LIN {X 768.326, Y -27.278, Z 404, A 0, B 90, C -0, E1 0, E2 0, E3 0, E4 0} C_DIS
LIN {X 766.132, Y -26.943, Z 404, A 0, B 90, C -0, E1 0, E2 0, E3 0, E4 0} C_DIS
LIN {X 763.95, Y -26.54, Z 404, A 0, B 90, C -0, E1 0, E2 0, E3 0, E4 0} C_DIS
LIN {X 761.781, Y -26.068, Z 404, A 0, B 90, C -0, E1 0, E2 0, E3 0, E4 0} C_DIS
LIN {X 759.629, Y -25.528, Z 404, A 0, B 90, C -0, E1 0, E2 0, E3 0, E4 0} C_DIS
LIN {X 757.494, Y -24.921, Z 404, A 0, B 90, C -0, E1 0, E2 0, E3 0, E4 0} C_DIS
LIN {X 755.379, Y -24.248, Z 404, A 0, B 90, C -0, E1 0, E2 0, E3 0, E4 0} C_DIS
LIN {X 753.287, Y -23.508, Z 404, A 0, B 90, C -0, E1 0, E2 0, E3 0, E4 0} C_DIS
LIN {X 751.219, Y -22.703, Z 404, A 0, B 90, C -0, E1 0, E2 0, E3 0, E4 0} C_DIS
LIN {X 749.177, Y -21.833, Z 404, A 0, B 90, C -0, E1 0, E2 0, E3 0, E4 0} C_DIS
LIN {X 747.163, Y -20.9, Z 404, A 0, B 90, C -0, E1 0, E2 0, E3 0, E4 0} C_DIS
LIN {X 745.18, Y -19.903, Z 404, A 0, B 90, C -0, E1 0, E2 0, E3 0, E4 0} C_DIS
LIN {X 743.229, Y -18.845, Z 404, A 0, B 90, C -0, E1 0, E2 0, E3 0, E4 0} C_DIS
LIN {X 741.313, Y -17.727, Z 404, A 0, B 90, C -0, E1 0, E2 0, E3 0, E4 0} C_DIS
LIN {X 739.432, Y -16.548, Z 404, A 0, B 90, C -0, E1 0, E2 0, E3 0, E4 0} C_DIS
LIN {X 737.589, Y -15.311, Z 404, A 0, B 90, C -0, E1 0, E2 0, E3 0, E4 0} C_DIS
LIN {X 735.786, Y -14.017, Z 404, A 0, B 90, C -0, E1 0, E2 0, E3 0, E4 0} C_DIS
LIN {X 734.025, Y -12.667, Z 404, A 0, B 90, C -0, E1 0, E2 0, E3 0, E4 0} C_DIS
LIN {X 732.307, Y -11.262, Z 404, A 0, B 90, C -0, E1 0, E2 0, E3 0, E4 0} C_DIS
LIN {X 730.634, Y -9.804, Z 404, A 0, B 90, C -0, E1 0, E2 0, E3 0, E4 0} C_DIS
LIN {X 729.007, Y -8.294, Z 404, A 0, B 90, C -0, E1 0, E2 0, E3 0, E4 0} C_DIS
LIN {X 727.429, Y -6.734, Z 404, A 0, B 90, C -0, E1 0, E2 0, E3 0, E4 0} C_DIS
LIN {X 725.901, Y -5.125, Z 404, A 0, B 90, C -0, E1 0, E2 0, E3 0, E4 0} C_DIS
LIN {X 724.423, Y -3.468, Z 404, A 0, B 90, C -0, E1 0, E2 0, E3 0, E4 0} C_DIS
LIN {X 722.999, Y -1.766, Z 404, A 0, B 90, C -0, E1 0, E2 0, E3 0, E4 0} C_DIS
LIN {X 721.629, Y -0.02, Z 404, A 0, B 90, C -0, E1 0, E2 0, E3 0, E4 0} C_DIS
LIN {X 720.314, Y 1.768, Z 404, A 0, B 90, C -0, E1 0, E2 0, E3 0, E4 0} C_DIS
LIN {X 719.056, Y 3.596, Z 404, A 0, B 90, C -0, E1 0, E2 0, E3 0, E4 0} C_DIS
LIN {X 717.856, Y 5.463, Z 404, A 0, B 90, C -0, E1 0, E2 0, E3 0, E4 0} C_DIS
LIN {X 716.715, Y 7.367, Z 404, A 0, B 90, C -0, E1 0, E2 0, E3 0, E4 0} C_DIS
LIN {X 715.635, Y 9.305, Z 404, A 0, B 90, C -0, E1 0, E2 0, E3 0, E4 0} C_DIS
LIN {X 714.616, Y 11.277, Z 404, A 0, B 90, C -0, E1 0, E2 0, E3 0, E4 0} C_DIS
LIN {X 713.66, Y 13.28, Z 404, A 0, B 90, C -0, E1 0, E2 0, E3 0, E4 0} C_DIS
LIN {X 712.767, Y 15.311, Z 404, A 0, B 90, C -0, E1 0, E2 0, E3 0, E4 0} C_DIS
LIN {X 711.938, Y 17.37, Z 404, A 0, B 90, C -0, E1 0, E2 0, E3 0, E4 0} C_DIS
LIN {X 711.174, Y 19.454, Z 404, A 0, B 90, C -0, E1 0, E2 0, E3 0, E4 0} C_DIS
LIN {X 710.476, Y 21.561, Z 404, A 0, B 90, C -0, E1 0, E2 0, E3 0, E4 0} C_DIS
LIN {X 709.845, Y 23.688, Z 404, A 0, B 90, C -0, E1 0, E2 0, E3 0, E4 0} C_DIS
LIN {X 709.281, Y 25.835, Z 404, A 0, B 90, C -0, E1 0, E2 0, E3 0, E4 0} C_DIS
LIN {X 708.784, Y 27.998, Z 404, A 0, B 90, C -0, E1 0, E2 0, E3 0, E4 0} C_DIS
LIN {X 708.356, Y 30.176, Z 404, A 0, B 90, C -0, E1 0, E2 0, E3 0, E4 0} C_DIS
LIN {X 707.996, Y 32.366, Z 404, A 0, B 90, C -0, E1 0, E2 0, E3 0, E4 0} C_DIS
LIN {X 707.705, Y 34.566, Z 404, A 0, B 90, C -0, E1 0, E2 0, E3 0, E4 0} C_DIS
LIN {X 707.484, Y 36.774, Z 404, A 0, B 90, C -0, E1 0, E2 0, E3 0, E4 0} C_DIS
LIN {X 707.332, Y 38.988, Z 404, A 0, B 90, C -0, E1 0, E2 0, E3 0, E4 0} C_DIS
LIN {X 707.25, Y 41.206, Z 404, A 0, B 90, C -0, E1 0, E2 0, E3 0, E4 0} C_DIS
LIN {X 707.237, Y 43.425, Z 404, A 0, B 90, C -0, E1 0, E2 0, E3 0, E4 0} C_DIS
LIN {X 707.294, Y 45.644, Z 404, A 0, B 90, C -0, E1 0, E2 0, E3 0, E4 0} C_DIS
LIN {X 707.42, Y 47.86, Z 404, A 0, B 90, C -0, E1 0, E2 0, E3 0, E4 0} C_DIS
LIN {X 707.617, Y 50.07, Z 404, A 0, B 90, C -0, E1 0, E2 0, E3 0, E4 0} C_DIS
LIN {X 707.882, Y 52.274, Z 404, A 0, B 90, C -0, E1 0, E2 0, E3 0, E4 0} C_DIS
LIN {X 708.217, Y 54.468, Z 404, A 0, B 90, C -0, E1 0, E2 0, E3 0, E4 0} C_DIS
LIN {X 708.62, Y 56.65, Z 404, A 0, B 90, C -0, E1 0, E2 0, E3 0, E4 0} C_DIS
LIN {X 709.092, Y 58.819, Z 404, A 0, B 90, C -0, E1 0, E2 0, E3 0, E4 0} C_DIS
LIN {X 709.632, Y 60.971, Z 404, A 0, B 90, C -0, E1 0, E2 0, E3 0, E4 0} C_DIS
LIN {X 710.239, Y 63.106, Z 404, A 0, B 90, C -0, E1 0, E2 0, E3 0, E4 0} C_DIS
LIN {X 710.912, Y 65.221, Z 404, A 0, B 90, C -0, E1 0, E2 0, E3 0, E4 0} C_DIS
LIN {X 711.828, Y 66.629, Z 406, A 0, B 90, C -0, E1 0, E2 0, E3 0, E4 0} C_DIS
LIN {X 712.612, Y 68.692, Z 406, A 0, B 90, C -0, E1 0, E2 0, E3 0, E4 0} C_DIS
LIN {X 713.46, Y 70.73, Z 406, A 0, B 90, C -0, E1 0, E2 0, E3 0, E4 0} C_DIS
LIN {X 714.371, Y 72.739, Z 406, A 0, B 90, C -0, E1 0, E2 0, E3 0, E4 0} C_DIS
LIN {X 715.346, Y 74.719, Z 406, A 0, B 90, C -0, E1 0, E2 0, E3 0, E4 0} C_DIS
LIN {X 716.382, Y 76.668, Z 406, A 0, B 90, C -0, E1 0, E2 0, E3 0, E4 0} C_DIS
LIN {X 717.478, Y 78.583, Z 406, A 0, B 90, C -0, E1 0, E2 0, E3 0, E4 0} C_DIS
LIN {X 718.635, Y 80.462, Z 406, A 0, B 90, C -0, E1 0, E2 0, E3 0, E4 0} C_DIS
LIN {X 719.849, Y 82.305, Z 406, A 0, B 90, C -0, E1 0, E2 0, E3 0, E4 0} C_DIS
LIN {X 721.121, Y 84.108, Z 406, A 0, B 90, C -0, E1 0, E2 0, E3 0, E4 0} C_DIS
LIN {X 722.449, Y 85.87, Z 406, A 0, B 90, C -0, E1 0, E2 0, E3 0, E4 0} C_DIS
LIN {X 723.832, Y 87.59, Z 406, A 0, B 90, C -0, E1 0, E2 0, E3 0, E4 0} C_DIS
LIN {X 725.268, Y 89.266, Z 406, A 0, B 90, C -0, E1 0, E2 0, E3 0, E4 0} C_DIS
LIN {X 726.756, Y 90.895, Z 406, A 0, B 90, C -0, E1 0, E2 0, E3 0, E4 0} C_DIS
LIN {X 728.295, Y 92.477, Z 406, A 0, B 90, C -0, E1 0, E2 0, E3 0, E4 0} C_DIS
LIN {X 729.882, Y 94.01, Z 406, A 0, B 90, C -0, E1 0, E2 0, E3 0, E4 0} C_DIS
LIN {X 731.517, Y 95.493, Z 406, A 0, B 90, C -0, E1 0, E2 0, E3 0, E4 0} C_DIS
LIN {X 733.197, Y 96.923, Z 406, A 0, B 90, C -0, E1 0, E2 0, E3 0, E4 0} C_DIS
LIN {X 734.922, Y 98.3, Z 406, A 0, B 90, C -0, E1 0, E2 0, E3 0, E4 0} C_DIS
LIN {X 736.689, Y 99.622, Z 406, A 0, B 90, C -0, E1 0, E2 0, E3 0, E4 0} C_DIS
LIN {X 738.496, Y 100.887, Z 406, A 0, B 90, C -0, E1 0, E2 0, E3 0, E4 0} C_DIS
LIN {X 740.343, Y 102.096, Z 406, A 0, B 90, C -0, E1 0, E2 0, E3 0, E4 0} C_DIS
LIN {X 742.227, Y 103.246, Z 406, A 0, B 90, C -0, E1 0, E2 0, E3 0, E4 0} C_DIS
LIN {X 744.145, Y 104.336, Z 406, A 0, B 90, C -0, E1 0, E2 0, E3 0, E4 0} C_DIS
LIN {X 746.097, Y 105.365, Z 406, A 0, B 90, C -0, E1 0, E2 0, E3 0, E4 0} C_DIS
LIN {X 748.081, Y 106.332, Z 406, A 0, B 90, C -0, E1 0, E2 0, E3 0, E4 0} C_DIS
LIN {X 750.094, Y 107.237, Z 406, A 0, B 90, C -0, E1 0, E2 0, E3 0, E4 0} C_DIS
LIN {X 752.134, Y 108.078, Z 406, A 0, B 90, C -0, E1 0, E2 0, E3 0, E4 0} C_DIS
LIN {X 754.199, Y 108.854, Z 406, A 0, B 90, C -0, E1 0, E2 0, E3 0, E4 0} C_DIS
LIN {X 756.288, Y 109.566, Z 406, A 0, B 90, C -0, E1 0, E2 0, E3 0, E4 0} C_DIS
LIN {X 758.399, Y 110.211, Z 406, A 0, B 90, C -0, E1 0, E2 0, E3 0, E4 0} C_DIS
LIN {X 760.528, Y 110.789, Z 406, A 0, B 90, C -0, E1 0, E2 0, E3 0, E4 0} C_DIS
LIN {X 762.675, Y 111.301, Z 406, A 0, B 90, C -0, E1 0, E2 0, E3 0, E4 0} C_DIS
LIN {X 764.837, Y 111.745, Z 406, A 0, B 90, C -0, E1 0, E2 0, E3 0, E4 0} C_DIS
LIN {X 767.011, Y 112.12, Z 406, A 0, B 90, C -0, E1 0, E2 0, E3 0, E4 0} C_DIS
LIN {X 769.197, Y 112.427, Z 406, A 0, B 90, C -0, E1 0, E2 0, E3 0, E4 0} C_DIS
LIN {X 771.39, Y 112.666, Z 406, A 0, B 90, C -0, E1 0, E2 0, E3 0, E4 0} C_DIS
LIN {X 773.591, Y 112.835, Z 406, A 0, B 90, C -0, E1 0, E2 0, E3 0, E4 0} C_DIS
LIN {X 775.795, Y 112.935, Z 406, A 0, B 90, C -0, E1 0, E2 0, E3 0, E4 0} C_DIS
LIN {X 778.002, Y 112.966, Z 406, A 0, B 90, C -0, E1 0, E2 0, E3 0, E4 0} C_DIS
LIN {X 780.208, Y 112.928, Z 406, A 0, B 90, C -0, E1 0, E2 0, E3 0, E4 0} C_DIS
LIN {X 782.412, Y 112.82, Z 406, A 0, B 90, C -0, E1 0, E2 0, E3 0, E4 0} C_DIS
LIN {X 784.612, Y 112.643, Z 406, A 0, B 90, C -0, E1 0, E2 0, E3 0, E4 0} C_DIS
LIN {X 786.805, Y 112.397, Z 406, A 0, B 90, C -0, E1 0, E2 0, E3 0, E4 0} C_DIS
LIN {X 788.989, Y 112.082, Z 406, A 0, B 90, C -0, E1 0, E2 0, E3 0, E4 0} C_DIS
LIN {X 791.162, Y 111.699, Z 406, A 0, B 90, C -0, E1 0, E2 0, E3 0, E4 0} C_DIS
LIN {X 793.322, Y 111.248, Z 406, A 0, B 90, C -0, E1 0, E2 0, E3 0, E4 0} C_DIS
LIN {X 795.467, Y 110.729, Z 406, A 0, B 90, C -0, E1 0, E2 0, E3 0, E4 0} C_DIS
LIN {X 797.595, Y 110.143, Z 406, A 0, B 90, C -0, E1 0, E2 0, E3 0, E4 0} C_DIS
LIN {X 799.703, Y 109.49, Z 406, A 0, B 90, C -0, E1 0, E2 0, E3 0, E4 0} C_DIS
LIN {X 801.789, Y 108.772, Z 406, A 0, B 90, C -0, E1 0, E2 0, E3 0, E4 0} C_DIS
LIN {X 803.852, Y 107.988, Z 406, A 0, B 90, C -0, E1 0, E2 0, E3 0, E4 0} C_DIS
LIN {X 805.89, Y 107.14, Z 406, A 0, B 90, C -0, E1 0, E2 0, E3 0, E4 0} C_DIS
LIN {X 807.899, Y 106.229, Z 406, A 0, B 90, C -0, E1 0, E2 0, E3 0, E4 0} C_DIS
LIN {X 809.879, Y 105.254, Z 406, A 0, B 90, C -0, E1 0, E2 0, E3 0, E4 0} C_DIS
LIN {X 811.828, Y 104.218, Z 406, A 0, B 90, C -0, E1 0, E2 0, E3 0, E4 0} C_DIS
LIN {X 813.743, Y 103.122, Z 406, A 0, B 90, C -0, E1 0, E2 0, E3 0, E4 0} C_DIS
LIN {X 815.622, Y 101.966, Z 406, A 0, B 90, C -0, E1 0, E2 0, E3 0, E4 0} C_DIS
LIN {X 817.465, Y 100.751, Z 406, A 0, B 90, C -0, E1 0, E2 0, E3 0, E4 0} C_DIS
LIN {X 819.268, Y 99.479, Z 406, A 0, B 90, C -0, E1 0, E2 0, E3 0, E4 0} C_DIS
LIN {X 821.03, Y 98.151, Z 406, A 0, B 90, C -0, E1 0, E2 0, E3 0, E4 0} C_DIS
LIN {X 822.75, Y 96.768, Z 406, A 0, B 90, C -0, E1 0, E2 0, E3 0, E4 0} C_DIS
LIN {X 824.426, Y 95.332, Z 406, A 0, B 90, C -0, E1 0, E2 0, E3 0, E4 0} C_DIS
LIN {X 826.055, Y 93.844, Z 406, A 0, B 90, C -0, E1 0, E2 0, E3 0, E4 0} C_DIS
LIN {X 827.637, Y 92.305, Z 406, A 0, B 90, C -0, E1 0, E2 0, E3 0, E4 0} C_DIS
LIN {X 829.17, Y 90.718, Z 406, A 0, B 90, C -0, E1 0, E2 0, E3 0, E4 0} C_DIS
LIN {X 830.653, Y 89.083, Z 406, A 0, B 90, C -0, E1 0, E2 0, E3 0, E4 0} C_DIS
LIN {X 832.083, Y 87.403, Z 406, A 0, B 90, C -0, E1 0, E2 0, E3 0, E4 0} C_DIS
LIN {X 833.46, Y 85.678, Z 406, A 0, B 90, C -0, E1 0, E2 0, E3 0, E4 0} C_DIS
LIN {X 834.782, Y 83.911, Z 406, A 0, B 90, C -0, E1 0, E2 0, E3 0, E4 0} C_DIS
LIN {X 836.047, Y 82.104, Z 406, A 0, B 90, C -0, E1 0, E2 0, E3 0, E4 0} C_DIS
LIN {X 837.256, Y 80.257, Z 406, A 0, B 90, C -0, E1 0, E2 0, E3 0, E4 0} C_DIS
LIN {X 838.406, Y 78.373, Z 406, A 0, B 90, C -0, E1 0, E2 0, E3 0, E4 0} C_DIS
LIN {X 839.496, Y 76.455, Z 406, A 0, B 90, C -0, E1 0, E2 0, E3 0, E4 0} C_DIS
LIN {X 840.525, Y 74.503, Z 406, A 0, B 90, C -0, E1 0, E2 0, E3 0, E4 0} C_DIS
LIN {X 841.492, Y 72.519, Z 406, A 0, B 90, C -0, E1 0, E2 0, E3 0, E4 0} C_DIS
LIN {X 842.397, Y 70.506, Z 406, A 0, B 90, C -0, E1 0, E2 0, E3 0, E4 0} C_DIS
LIN {X 843.238, Y 68.466, Z 406, A 0, B 90, C -0, E1 0, E2 0, E3 0, E4 0} C_DIS
LIN {X 844.014, Y 66.401, Z 406, A 0, B 90, C -0, E1 0, E2 0, E3 0, E4 0} C_DIS
LIN {X 844.726, Y 64.312, Z 406, A 0, B 90, C -0, E1 0, E2 0, E3 0, E4 0} C_DIS
LIN {X 845.371, Y 62.201, Z 406, A 0, B 90, C -0, E1 0, E2 0, E3 0, E4 0} C_DIS
LIN {X 845.949, Y 60.072, Z 406, A 0, B 90, C -0, E1 0, E2 0, E3 0, E4 0} C_DIS
LIN {X 846.461, Y 57.925, Z 406, A 0, B 90, C -0, E1 0, E2 0, E3 0, E4 0} C_DIS
LIN {X 846.905, Y 55.763, Z 406, A 0, B 90, C -0, E1 0, E2 0, E3 0, E4 0} C_DIS
LIN {X 847.28, Y 53.589, Z 406, A 0, B 90, C -0, E1 0, E2 0, E3 0, E4 0} C_DIS
LIN {X 847.587, Y 51.403, Z 406, A 0, B 90, C -0, E1 0, E2 0, E3 0, E4 0} C_DIS
LIN {X 847.826, Y 49.21, Z 406, A 0, B 90, C -0, E1 0, E2 0, E3 0, E4 0} C_DIS
LIN {X 847.995, Y 47.009, Z 406, A 0, B 90, C -0, E1 0, E2 0, E3 0, E4 0} C_DIS
LIN {X 848.095, Y 44.805, Z 406, A 0, B 90, C -0, E1 0, E2 0, E3 0, E4 0} C_DIS
LIN {X 848.126, Y 42.598, Z 406, A 0, B 90, C -0, E1 0, E2 0, E3 0, E4 0} C_DIS
LIN {X 848.088, Y 40.392, Z 406, A 0, B 90, C -0, E1 0, E2 0, E3 0, E4 0} C_DIS
LIN {X 847.98, Y 38.188, Z 406, A 0, B 90, C -0, E1 0, E2 0, E3 0, E4 0} C_DIS
LIN {X 847.803, Y 35.988, Z 406, A 0, B 90, C -0, E1 0, E2 0, E3 0, E4 0} C_DIS
LIN {X 847.557, Y 33.795, Z 406, A 0, B 90, C -0, E1 0, E2 0, E3 0, E4 0} C_DIS
LIN {X 847.242, Y 31.611, Z 406, A 0, B 90, C -0, E1 0, E2 0, E3 0, E4 0} C_DIS
LIN {X 846.859, Y 29.438, Z 406, A 0, B 90, C -0, E1 0, E2 0, E3 0, E4 0} C_DIS
LIN {X 846.408, Y 27.278, Z 406, A 0, B 90, C -0, E1 0, E2 0, E3 0, E4 0} C_DIS
LIN {X 845.889, Y 25.133, Z 406, A 0, B 90, C -0, E1 0, E2 0, E3 0, E4 0} C_DIS
LIN {X 845.303, Y 23.005, Z 406, A 0, B 90, C -0, E1 0, E2 0, E3 0, E4 0} C_DIS
LIN {X 844.65, Y 20.897, Z 406, A 0, B 90, C -0, E1 0, E2 0, E3 0, E4 0} C_DIS
LIN {X 843.932, Y 18.811, Z 406, A 0, B 90, C -0, E1 0, E2 0, E3 0, E4 0} C_DIS
LIN {X 843.148, Y 16.748, Z 406, A 0, B 90, C -0, E1 0, E2 0, E3 0, E4 0} C_DIS
LIN {X 842.3, Y 14.71, Z 406, A 0, B 90, C -0, E1 0, E2 0, E3 0, E4 0} C_DIS
LIN {X 841.389, Y 12.701, Z 406, A 0, B 90, C -0, E1 0, E2 0, E3 0, E4 0} C_DIS
LIN {X 840.414, Y 10.721, Z 406, A 0, B 90, C -0, E1 0, E2 0, E3 0, E4 0} C_DIS
LIN {X 839.378, Y 8.772, Z 406, A 0, B 90, C -0, E1 0, E2 0, E3 0, E4 0} C_DIS
LIN {X 838.282, Y 6.857, Z 406, A 0, B 90, C -0, E1 0, E2 0, E3 0, E4 0} C_DIS
LIN {X 837.125, Y 4.978, Z 406, A 0, B 90, C -0, E1 0, E2 0, E3 0, E4 0} C_DIS
LIN {X 835.911, Y 3.135, Z 406, A 0, B 90, C -0, E1 0, E2 0, E3 0, E4 0} C_DIS
LIN {X 834.639, Y 1.332, Z 406, A 0, B 90, C -0, E1 0, E2 0, E3 0, E4 0} C_DIS
LIN {X 833.311, Y -0.43, Z 406, A 0, B 90, C -0, E1 0, E2 0, E3 0, E4 0} C_DIS
LIN {X 831.928, Y -2.15, Z 406, A 0, B 90, C -0, E1 0, E2 0, E3 0, E4 0} C_DIS
LIN {X 830.492, Y -3.826, Z 406, A 0, B 90, C -0, E1 0, E2 0, E3 0, E4 0} C_DIS
LIN {X 829.004, Y -5.455, Z 406, A 0, B 90, C -0, E1 0, E2 0, E3 0, E4 0} C_DIS
LIN {X 827.465, Y -7.037, Z 406, A 0, B 90, C -0, E1 0, E2 0, E3 0, E4 0} C_DIS
LIN {X 825.878, Y -8.57, Z 406, A 0, B 90, C -0, E1 0, E2 0, E3 0, E4 0} C_DIS
LIN {X 824.243, Y -10.053, Z 406, A 0, B 90, C -0, E1 0, E2 0, E3 0, E4 0} C_DIS
LIN {X 822.563, Y -11.483, Z 406, A 0, B 90, C -0, E1 0, E2 0, E3 0, E4 0} C_DIS
LIN {X 820.838, Y -12.86, Z 406, A 0, B 90, C -0, E1 0, E2 0, E3 0, E4 0} C_DIS
LIN {X 819.071, Y -14.182, Z 406, A 0, B 90, C -0, E1 0, E2 0, E3 0, E4 0} C_DIS
LIN {X 817.263, Y -15.447, Z 406, A 0, B 90, C -0, E1 0, E2 0, E3 0, E4 0} C_DIS
LIN {X 815.417, Y -16.656, Z 406, A 0, B 90, C -0, E1 0, E2 0, E3 0, E4 0} C_DIS
LIN {X 813.533, Y -17.806, Z 406, A 0, B 90, C -0, E1 0, E2 0, E3 0, E4 0} C_DIS
LIN {X 811.615, Y -18.896, Z 406, A 0, B 90, C -0, E1 0, E2 0, E3 0, E4 0} C_DIS
LIN {X 809.663, Y -19.925, Z 406, A 0, B 90, C -0, E1 0, E2 0, E3 0, E4 0} C_DIS
LIN {X 807.679, Y -20.892, Z 406, A 0, B 90, C -0, E1 0, E2 0, E3 0, E4 0} C_DIS
LIN {X 805.666, Y -21.797, Z 406, A 0, B 90, C -0, E1 0, E2 0, E3 0, E4 0} C_DIS
LIN {X 803.626, Y -22.638, Z 406, A 0, B 90, C -0, E1 0, E2 0, E3 0, E4 0} C_DIS
LIN {X 801.561, Y -23.414, Z 406, A 0, B 90, C -0, E1 0, E2 0, E3 0, E4 0} C_DIS
LIN {X 799.471, Y -24.126, Z 406, A 0, B 90, C -0, E1 0, E2 0, E3 0, E4 0} C_DIS
LIN {X 797.361, Y -24.771, Z 406, A 0, B 90, C -0, E1 0, E2 0, E3 0, E4 0} C_DIS
LIN {X 795.232, Y -25.349, Z 406, A 0, B 90, C -0, E1 0, E2 0, E3 0, E4 0} C_DIS
LIN {X 793.085, Y -25.861, Z 406, A 0, B 90, C -0, E1 0, E2 0, E3 0, E4 0} C_DIS
LIN {X 790.923, Y -26.305, Z 406, A 0, B 90, C -0, E1 0, E2 0, E3 0, E4 0} C_DIS
LIN {X 788.749, Y -26.68, Z 406, A 0, B 90, C -0, E1 0, E2 0, E3 0, E4 0} C_DIS
LIN {X 786.563, Y -26.987, Z 406, A 0, B 90, C -0, E1 0, E2 0, E3 0, E4 0} C_DIS
LIN {X 784.37, Y -27.226, Z 406, A 0, B 90, C -0, E1 0, E2 0, E3 0, E4 0} C_DIS
LIN {X 782.169, Y -27.395, Z 406, A 0, B 90, C -0, E1 0, E2 0, E3 0, E4 0} C_DIS
LIN {X 779.965, Y -27.495, Z 406, A 0, B 90, C -0, E1 0, E2 0, E3 0, E4 0} C_DIS
LIN {X 777.758, Y -27.526, Z 406, A 0, B 90, C -0, E1 0, E2 0, E3 0, E4 0} C_DIS
LIN {X 775.552, Y -27.488, Z 406, A 0, B 90, C -0, E1 0, E2 0, E3 0, E4 0} C_DIS
LIN {X 773.348, Y -27.38, Z 406, A 0, B 90, C -0, E1 0, E2 0, E3 0, E4 0} C_DIS
LIN {X 771.148, Y -27.203, Z 406, A 0, B 90, C -0, E1 0, E2 0, E3 0, E4 0} C_DIS
LIN {X 768.955, Y -26.957, Z 406, A 0, B 90, C -0, E1 0, E2 0, E3 0, E4 0} C_DIS
LIN {X 766.771, Y -26.642, Z 406, A 0, B 90, C -0, E1 0, E2 0, E3 0, E4 0} C_DIS
LIN {X 764.598, Y -26.259, Z 406, A 0, B 90, C -0, E1 0, E2 0, E3 0, E4 0} C_DIS
LIN {X 762.438, Y -25.808, Z 406, A 0, B 90, C -0, E1 0, E2 0, E3 0, E4 0} C_DIS
LIN {X 760.293, Y -25.289, Z 406, A 0, B 90, C -0, E1 0, E2 0, E3 0, E4 0} C_DIS
LIN {X 758.165, Y -24.703, Z 406, A 0, B 90, C -0, E1 0, E2 0, E3 0, E4 0} C_DIS
LIN {X 756.057, Y -24.05, Z 406, A 0, B 90, C -0, E1 0, E2 0, E3 0, E4 0} C_DIS
LIN {X 753.971, Y -23.332, Z 406, A 0, B 90, C -0, E1 0, E2 0, E3 0, E4 0} C_DIS
LIN {X 751.908, Y -22.548, Z 406, A 0, B 90, C -0, E1 0, E2 0, E3 0, E4 0} C_DIS
LIN {X 749.87, Y -21.7, Z 406, A 0, B 90, C -0, E1 0, E2 0, E3 0, E4 0} C_DIS
LIN {X 747.861, Y -20.789, Z 406, A 0, B 90, C -0, E1 0, E2 0, E3 0, E4 0} C_DIS
LIN {X 745.881, Y -19.814, Z 406, A 0, B 90, C -0, E1 0, E2 0, E3 0, E4 0} C_DIS
LIN {X 743.932, Y -18.778, Z 406, A 0, B 90, C -0, E1 0, E2 0, E3 0, E4 0} C_DIS
LIN {X 742.017, Y -17.682, Z 406, A 0, B 90, C -0, E1 0, E2 0, E3 0, E4 0} C_DIS
LIN {X 740.138, Y -16.526, Z 406, A 0, B 90, C -0, E1 0, E2 0, E3 0, E4 0} C_DIS
LIN {X 738.295, Y -15.311, Z 406, A 0, B 90, C -0, E1 0, E2 0, E3 0, E4 0} C_DIS
LIN {X 736.492, Y -14.039, Z 406, A 0, B 90, C -0, E1 0, E2 0, E3 0, E4 0} C_DIS
LIN {X 734.73, Y -12.711, Z 406, A 0, B 90, C -0, E1 0, E2 0, E3 0, E4 0} C_DIS
LIN {X 733.01, Y -11.328, Z 406, A 0, B 90, C -0, E1 0, E2 0, E3 0, E4 0} C_DIS
LIN {X 731.334, Y -9.892, Z 406, A 0, B 90, C -0, E1 0, E2 0, E3 0, E4 0} C_DIS
LIN {X 729.705, Y -8.404, Z 406, A 0, B 90, C -0, E1 0, E2 0, E3 0, E4 0} C_DIS
LIN {X 728.123, Y -6.865, Z 406, A 0, B 90, C -0, E1 0, E2 0, E3 0, E4 0} C_DIS
LIN {X 726.59, Y -5.278, Z 406, A 0, B 90, C -0, E1 0, E2 0, E3 0, E4 0} C_DIS
LIN {X 725.107, Y -3.643, Z 406, A 0, B 90, C -0, E1 0, E2 0, E3 0, E4 0} C_DIS
LIN {X 723.677, Y -1.963, Z 406, A 0, B 90, C -0, E1 0, E2 0, E3 0, E4 0} C_DIS
LIN {X 722.3, Y -0.238, Z 406, A 0, B 90, C -0, E1 0, E2 0, E3 0, E4 0} C_DIS
LIN {X 720.978, Y 1.529, Z 406, A 0, B 90, C -0, E1 0, E2 0, E3 0, E4 0} C_DIS
LIN {X 719.713, Y 3.336, Z 406, A 0, B 90, C -0, E1 0, E2 0, E3 0, E4 0} C_DIS
LIN {X 718.504, Y 5.183, Z 406, A 0, B 90, C -0, E1 0, E2 0, E3 0, E4 0} C_DIS
LIN {X 717.354, Y 7.067, Z 406, A 0, B 90, C -0, E1 0, E2 0, E3 0, E4 0} C_DIS
LIN {X 716.264, Y 8.985, Z 406, A 0, B 90, C -0, E1 0, E2 0, E3 0, E4 0} C_DIS
LIN {X 715.235, Y 10.937, Z 406, A 0, B 90, C -0, E1 0, E2 0, E3 0, E4 0} C_DIS
LIN {X 714.268, Y 12.921, Z 406, A 0, B 90, C -0, E1 0, E2 0, E3 0, E4 0} C_DIS
LIN {X 713.363, Y 14.934, Z 406, A 0, B 90, C -0, E1 0, E2 0, E3 0, E4 0} C_DIS
LIN {X 712.522, Y 16.974, Z 406, A 0, B 90, C -0, E1 0, E2 0, E3 0, E4 0} C_DIS
LIN {X 711.746, Y 19.039, Z 406, A 0, B 90, C -0, E1 0, E2 0, E3 0, E4 0} C_DIS
LIN {X 711.034, Y 21.128, Z 406, A 0, B 90, C -0, E1 0, E2 0, E3 0, E4 0} C_DIS
LIN {X 710.389, Y 23.239, Z 406, A 0, B 90, C -0, E1 0, E2 0, E3 0, E4 0} C_DIS
LIN {X 709.811, Y 25.368, Z 406, A 0, B 90, C -0, E1 0, E2 0, E3 0, E4 0} C_DIS
LIN {X 709.299, Y 27.515, Z 406, A 0, B 90, C -0, E1 0, E2 0, E3 0, E4 0} C_DIS
LIN {X 708.855, Y 29.677, Z 406, A 0, B 90, C -0, E1 0, E2 0, E3 0, E4 0} C_DIS
LIN {X 708.48, Y 31.851, Z 406, A 0, B 90, C -0, E1 0, E2 0, E3 0, E4 0} C_DIS
LIN {X 708.173, Y 34.037, Z 406, A 0, B 90, C -0, E1 0, E2 0, E3 0, E4 0} C_DIS
LIN {X 707.934, Y 36.23, Z 406, A 0, B 90, C -0, E1 0, E2 0, E3 0, E4 0} C_DIS
LIN {X 707.765, Y 38.431, Z 406, A 0, B 90, C -0, E1 0, E2 0, E3 0, E4 0} C_DIS
LIN {X 707.665, Y 40.635, Z 406, A 0, B 90, C -0, E1 0, E2 0, E3 0, E4 0} C_DIS
LIN {X 707.634, Y 42.842, Z 406, A 0, B 90, C -0, E1 0, E2 0, E3 0, E4 0} C_DIS
LIN {X 707.672, Y 45.048, Z 406, A 0, B 90, C -0, E1 0, E2 0, E3 0, E4 0} C_DIS
LIN {X 707.78, Y 47.252, Z 406, A 0, B 90, C -0, E1 0, E2 0, E3 0, E4 0} C_DIS
LIN {X 707.957, Y 49.452, Z 406, A 0, B 90, C -0, E1 0, E2 0, E3 0, E4 0} C_DIS
LIN {X 708.203, Y 51.645, Z 406, A 0, B 90, C -0, E1 0, E2 0, E3 0, E4 0} C_DIS
LIN {X 708.518, Y 53.829, Z 406, A 0, B 90, C -0, E1 0, E2 0, E3 0, E4 0} C_DIS
LIN {X 708.901, Y 56.002, Z 406, A 0, B 90, C -0, E1 0, E2 0, E3 0, E4 0} C_DIS
LIN {X 709.352, Y 58.162, Z 406, A 0, B 90, C -0, E1 0, E2 0, E3 0, E4 0} C_DIS
LIN {X 709.871, Y 60.307, Z 406, A 0, B 90, C -0, E1 0, E2 0, E3 0, E4 0} C_DIS
LIN {X 710.457, Y 62.435, Z 406, A 0, B 90, C -0, E1 0, E2 0, E3 0, E4 0} C_DIS
LIN {X 711.11, Y 64.543, Z 406, A 0, B 90, C -0, E1 0, E2 0, E3 0, E4 0} C_DIS
LIN {X 712.009, Y 65.962, Z 408, A 0, B 90, C -0, E1 0, E2 0, E3 0, E4 0} C_DIS
LIN {X 712.771, Y 68.02, Z 408, A 0, B 90, C -0, E1 0, E2 0, E3 0, E4 0} C_DIS
LIN {X 713.598, Y 70.052, Z 408, A 0, B 90, C -0, E1 0, E2 0, E3 0, E4 0} C_DIS
LIN {X 714.488, Y 72.058, Z 408, A 0, B 90, C -0, E1 0, E2 0, E3 0, E4 0} C_DIS
LIN {X 715.441, Y 74.035, Z 408, A 0, B 90, C -0, E1 0, E2 0, E3 0, E4 0} C_DIS
LIN {X 716.455, Y 75.98, Z 408, A 0, B 90, C -0, E1 0, E2 0, E3 0, E4 0} C_DIS
LIN {X 717.53, Y 77.893, Z 408, A 0, B 90, C -0, E1 0, E2 0, E3 0, E4 0} C_DIS
LIN {X 718.665, Y 79.772, Z 408, A 0, B 90, C -0, E1 0, E2 0, E3 0, E4 0} C_DIS
LIN {X 719.858, Y 81.613, Z 408, A 0, B 90, C -0, E1 0, E2 0, E3 0, E4 0} C_DIS
LIN {X 721.108, Y 83.417, Z 408, A 0, B 90, C -0, E1 0, E2 0, E3 0, E4 0} C_DIS
LIN {X 722.415, Y 85.18, Z 408, A 0, B 90, C -0, E1 0, E2 0, E3 0, E4 0} C_DIS
LIN {X 723.776, Y 86.901, Z 408, A 0, B 90, C -0, E1 0, E2 0, E3 0, E4 0} C_DIS
LIN {X 725.19, Y 88.579, Z 408, A 0, B 90, C -0, E1 0, E2 0, E3 0, E4 0} C_DIS
LIN {X 726.657, Y 90.211, Z 408, A 0, B 90, C -0, E1 0, E2 0, E3 0, E4 0} C_DIS
LIN {X 728.174, Y 91.797, Z 408, A 0, B 90, C -0, E1 0, E2 0, E3 0, E4 0} C_DIS
LIN {X 729.74, Y 93.334, Z 408, A 0, B 90, C -0, E1 0, E2 0, E3 0, E4 0} C_DIS
LIN {X 731.353, Y 94.821, Z 408, A 0, B 90, C -0, E1 0, E2 0, E3 0, E4 0} C_DIS
LIN {X 733.013, Y 96.257, Z 408, A 0, B 90, C -0, E1 0, E2 0, E3 0, E4 0} C_DIS
LIN {X 734.717, Y 97.64, Z 408, A 0, B 90, C -0, E1 0, E2 0, E3 0, E4 0} C_DIS
LIN {X 736.463, Y 98.968, Z 408, A 0, B 90, C -0, E1 0, E2 0, E3 0, E4 0} C_DIS
LIN {X 738.25, Y 100.242, Z 408, A 0, B 90, C -0, E1 0, E2 0, E3 0, E4 0} C_DIS
LIN {X 740.077, Y 101.458, Z 408, A 0, B 90, C -0, E1 0, E2 0, E3 0, E4 0} C_DIS
LIN {X 741.94, Y 102.616, Z 408, A 0, B 90, C -0, E1 0, E2 0, E3 0, E4 0} C_DIS
LIN {X 743.839, Y 103.716, Z 408, A 0, B 90, C -0, E1 0, E2 0, E3 0, E4 0} C_DIS
LIN {X 745.772, Y 104.755, Z 408, A 0, B 90, C -0, E1 0, E2 0, E3 0, E4 0} C_DIS
LIN {X 747.736, Y 105.733, Z 408, A 0, B 90, C -0, E1 0, E2 0, E3 0, E4 0} C_DIS
LIN {X 749.731, Y 106.649, Z 408, A 0, B 90, C -0, E1 0, E2 0, E3 0, E4 0} C_DIS
LIN {X 751.753, Y 107.501, Z 408, A 0, B 90, C -0, E1 0, E2 0, E3 0, E4 0} C_DIS
LIN {X 753.8, Y 108.29, Z 408, A 0, B 90, C -0, E1 0, E2 0, E3 0, E4 0} C_DIS
LIN {X 755.872, Y 109.014, Z 408, A 0, B 90, C -0, E1 0, E2 0, E3 0, E4 0} C_DIS
LIN {X 757.965, Y 109.672, Z 408, A 0, B 90, C -0, E1 0, E2 0, E3 0, E4 0} C_DIS
LIN {X 760.078, Y 110.265, Z 408, A 0, B 90, C -0, E1 0, E2 0, E3 0, E4 0} C_DIS
LIN {X 762.208, Y 110.791, Z 408, A 0, B 90, C -0, E1 0, E2 0, E3 0, E4 0} C_DIS
LIN {X 764.354, Y 111.25, Z 408, A 0, B 90, C -0, E1 0, E2 0, E3 0, E4 0} C_DIS
LIN {X 766.513, Y 111.641, Z 408, A 0, B 90, C -0, E1 0, E2 0, E3 0, E4 0} C_DIS
LIN {X 768.684, Y 111.964, Z 408, A 0, B 90, C -0, E1 0, E2 0, E3 0, E4 0} C_DIS
LIN {X 770.863, Y 112.218, Z 408, A 0, B 90, C -0, E1 0, E2 0, E3 0, E4 0} C_DIS
LIN {X 773.05, Y 112.404, Z 408, A 0, B 90, C -0, E1 0, E2 0, E3 0, E4 0} C_DIS
LIN {X 775.241, Y 112.522, Z 408, A 0, B 90, C -0, E1 0, E2 0, E3 0, E4 0} C_DIS
LIN {X 777.435, Y 112.57, Z 408, A 0, B 90, C -0, E1 0, E2 0, E3 0, E4 0} C_DIS
LIN {X 779.629, Y 112.55, Z 408, A 0, B 90, C -0, E1 0, E2 0, E3 0, E4 0} C_DIS
LIN {X 781.822, Y 112.46, Z 408, A 0, B 90, C -0, E1 0, E2 0, E3 0, E4 0} C_DIS
LIN {X 784.01, Y 112.302, Z 408, A 0, B 90, C -0, E1 0, E2 0, E3 0, E4 0} C_DIS
LIN {X 786.193, Y 112.075, Z 408, A 0, B 90, C -0, E1 0, E2 0, E3 0, E4 0} C_DIS
LIN {X 788.367, Y 111.78, Z 408, A 0, B 90, C -0, E1 0, E2 0, E3 0, E4 0} C_DIS
LIN {X 790.531, Y 111.416, Z 408, A 0, B 90, C -0, E1 0, E2 0, E3 0, E4 0} C_DIS
LIN {X 792.683, Y 110.985, Z 408, A 0, B 90, C -0, E1 0, E2 0, E3 0, E4 0} C_DIS
LIN {X 794.82, Y 110.486, Z 408, A 0, B 90, C -0, E1 0, E2 0, E3 0, E4 0} C_DIS
LIN {X 796.94, Y 109.921, Z 408, A 0, B 90, C -0, E1 0, E2 0, E3 0, E4 0} C_DIS
LIN {X 799.042, Y 109.289, Z 408, A 0, B 90, C -0, E1 0, E2 0, E3 0, E4 0} C_DIS
LIN {X 801.122, Y 108.591, Z 408, A 0, B 90, C -0, E1 0, E2 0, E3 0, E4 0} C_DIS
LIN {X 803.18, Y 107.829, Z 408, A 0, B 90, C -0, E1 0, E2 0, E3 0, E4 0} C_DIS
LIN {X 805.212, Y 107.002, Z 408, A 0, B 90, C -0, E1 0, E2 0, E3 0, E4 0} C_DIS
LIN {X 807.218, Y 106.112, Z 408, A 0, B 90, C -0, E1 0, E2 0, E3 0, E4 0} C_DIS
LIN {X 809.195, Y 105.159, Z 408, A 0, B 90, C -0, E1 0, E2 0, E3 0, E4 0} C_DIS
LIN {X 811.141, Y 104.145, Z 408, A 0, B 90, C -0, E1 0, E2 0, E3 0, E4 0} C_DIS
LIN {X 813.053, Y 103.07, Z 408, A 0, B 90, C -0, E1 0, E2 0, E3 0, E4 0} C_DIS
LIN {X 814.932, Y 101.935, Z 408, A 0, B 90, C -0, E1 0, E2 0, E3 0, E4 0} C_DIS
LIN {X 816.773, Y 100.742, Z 408, A 0, B 90, C -0, E1 0, E2 0, E3 0, E4 0} C_DIS
LIN {X 818.577, Y 99.492, Z 408, A 0, B 90, C -0, E1 0, E2 0, E3 0, E4 0} C_DIS
LIN {X 820.34, Y 98.185, Z 408, A 0, B 90, C -0, E1 0, E2 0, E3 0, E4 0} C_DIS
LIN {X 822.061, Y 96.824, Z 408, A 0, B 90, C -0, E1 0, E2 0, E3 0, E4 0} C_DIS
LIN {X 823.739, Y 95.41, Z 408, A 0, B 90, C -0, E1 0, E2 0, E3 0, E4 0} C_DIS
LIN {X 825.371, Y 93.943, Z 408, A 0, B 90, C -0, E1 0, E2 0, E3 0, E4 0} C_DIS
LIN {X 826.957, Y 92.426, Z 408, A 0, B 90, C -0, E1 0, E2 0, E3 0, E4 0} C_DIS
LIN {X 828.494, Y 90.86, Z 408, A 0, B 90, C -0, E1 0, E2 0, E3 0, E4 0} C_DIS
LIN {X 829.981, Y 89.247, Z 408, A 0, B 90, C -0, E1 0, E2 0, E3 0, E4 0} C_DIS
LIN {X 831.417, Y 87.587, Z 408, A 0, B 90, C -0, E1 0, E2 0, E3 0, E4 0} C_DIS
LIN {X 832.8, Y 85.883, Z 408, A 0, B 90, C -0, E1 0, E2 0, E3 0, E4 0} C_DIS
LIN {X 834.128, Y 84.137, Z 408, A 0, B 90, C -0, E1 0, E2 0, E3 0, E4 0} C_DIS
LIN {X 835.401, Y 82.35, Z 408, A 0, B 90, C -0, E1 0, E2 0, E3 0, E4 0} C_DIS
LIN {X 836.618, Y 80.523, Z 408, A 0, B 90, C -0, E1 0, E2 0, E3 0, E4 0} C_DIS
LIN {X 837.776, Y 78.66, Z 408, A 0, B 90, C -0, E1 0, E2 0, E3 0, E4 0} C_DIS
LIN {X 838.876, Y 76.761, Z 408, A 0, B 90, C -0, E1 0, E2 0, E3 0, E4 0} C_DIS
LIN {X 839.915, Y 74.828, Z 408, A 0, B 90, C -0, E1 0, E2 0, E3 0, E4 0} C_DIS
LIN {X 840.893, Y 72.864, Z 408, A 0, B 90, C -0, E1 0, E2 0, E3 0, E4 0} C_DIS
LIN {X 841.809, Y 70.869, Z 408, A 0, B 90, C -0, E1 0, E2 0, E3 0, E4 0} C_DIS
LIN {X 842.661, Y 68.847, Z 408, A 0, B 90, C -0, E1 0, E2 0, E3 0, E4 0} C_DIS
LIN {X 843.45, Y 66.8, Z 408, A 0, B 90, C -0, E1 0, E2 0, E3 0, E4 0} C_DIS
LIN {X 844.174, Y 64.728, Z 408, A 0, B 90, C -0, E1 0, E2 0, E3 0, E4 0} C_DIS
LIN {X 844.832, Y 62.635, Z 408, A 0, B 90, C -0, E1 0, E2 0, E3 0, E4 0} C_DIS
LIN {X 845.425, Y 60.522, Z 408, A 0, B 90, C -0, E1 0, E2 0, E3 0, E4 0} C_DIS
LIN {X 845.951, Y 58.392, Z 408, A 0, B 90, C -0, E1 0, E2 0, E3 0, E4 0} C_DIS
LIN {X 846.409, Y 56.246, Z 408, A 0, B 90, C -0, E1 0, E2 0, E3 0, E4 0} C_DIS
LIN {X 846.801, Y 54.087, Z 408, A 0, B 90, C -0, E1 0, E2 0, E3 0, E4 0} C_DIS
LIN {X 847.124, Y 51.916, Z 408, A 0, B 90, C -0, E1 0, E2 0, E3 0, E4 0} C_DIS
LIN {X 847.378, Y 49.737, Z 408, A 0, B 90, C -0, E1 0, E2 0, E3 0, E4 0} C_DIS
LIN {X 847.564, Y 47.55, Z 408, A 0, B 90, C -0, E1 0, E2 0, E3 0, E4 0} C_DIS
LIN {X 847.682, Y 45.359, Z 408, A 0, B 90, C -0, E1 0, E2 0, E3 0, E4 0} C_DIS
LIN {X 847.73, Y 43.165, Z 408, A 0, B 90, C -0, E1 0, E2 0, E3 0, E4 0} C_DIS
LIN {X 847.71, Y 40.971, Z 408, A 0, B 90, C -0, E1 0, E2 0, E3 0, E4 0} C_DIS
LIN {X 847.62, Y 38.778, Z 408, A 0, B 90, C -0, E1 0, E2 0, E3 0, E4 0} C_DIS
LIN {X 847.462, Y 36.59, Z 408, A 0, B 90, C -0, E1 0, E2 0, E3 0, E4 0} C_DIS
LIN {X 847.235, Y 34.407, Z 408, A 0, B 90, C -0, E1 0, E2 0, E3 0, E4 0} C_DIS
LIN {X 846.94, Y 32.233, Z 408, A 0, B 90, C -0, E1 0, E2 0, E3 0, E4 0} C_DIS
LIN {X 846.576, Y 30.069, Z 408, A 0, B 90, C -0, E1 0, E2 0, E3 0, E4 0} C_DIS
LIN {X 846.145, Y 27.917, Z 408, A 0, B 90, C -0, E1 0, E2 0, E3 0, E4 0} C_DIS
LIN {X 845.646, Y 25.78, Z 408, A 0, B 90, C -0, E1 0, E2 0, E3 0, E4 0} C_DIS
LIN {X 845.081, Y 23.66, Z 408, A 0, B 90, C -0, E1 0, E2 0, E3 0, E4 0} C_DIS
LIN {X 844.449, Y 21.558, Z 408, A 0, B 90, C -0, E1 0, E2 0, E3 0, E4 0} C_DIS
LIN {X 843.751, Y 19.478, Z 408, A 0, B 90, C -0, E1 0, E2 0, E3 0, E4 0} C_DIS
LIN {X 842.989, Y 17.42, Z 408, A 0, B 90, C -0, E1 0, E2 0, E3 0, E4 0} C_DIS
LIN {X 842.162, Y 15.388, Z 408, A 0, B 90, C -0, E1 0, E2 0, E3 0, E4 0} C_DIS
LIN {X 841.272, Y 13.382, Z 408, A 0, B 90, C -0, E1 0, E2 0, E3 0, E4 0} C_DIS
LIN {X 840.319, Y 11.405, Z 408, A 0, B 90, C -0, E1 0, E2 0, E3 0, E4 0} C_DIS
LIN {X 839.305, Y 9.46, Z 408, A 0, B 90, C -0, E1 0, E2 0, E3 0, E4 0} C_DIS
LIN {X 838.23, Y 7.547, Z 408, A 0, B 90, C -0, E1 0, E2 0, E3 0, E4 0} C_DIS
LIN {X 837.095, Y 5.668, Z 408, A 0, B 90, C -0, E1 0, E2 0, E3 0, E4 0} C_DIS
LIN {X 835.902, Y 3.827, Z 408, A 0, B 90, C -0, E1 0, E2 0, E3 0, E4 0} C_DIS
LIN {X 834.652, Y 2.023, Z 408, A 0, B 90, C -0, E1 0, E2 0, E3 0, E4 0} C_DIS
LIN {X 833.345, Y 0.26, Z 408, A 0, B 90, C -0, E1 0, E2 0, E3 0, E4 0} C_DIS
LIN {X 831.984, Y -1.461, Z 408, A 0, B 90, C -0, E1 0, E2 0, E3 0, E4 0} C_DIS
LIN {X 830.57, Y -3.139, Z 408, A 0, B 90, C -0, E1 0, E2 0, E3 0, E4 0} C_DIS
LIN {X 829.103, Y -4.771, Z 408, A 0, B 90, C -0, E1 0, E2 0, E3 0, E4 0} C_DIS
LIN {X 827.586, Y -6.357, Z 408, A 0, B 90, C -0, E1 0, E2 0, E3 0, E4 0} C_DIS
LIN {X 826.02, Y -7.894, Z 408, A 0, B 90, C -0, E1 0, E2 0, E3 0, E4 0} C_DIS
LIN {X 824.407, Y -9.381, Z 408, A 0, B 90, C -0, E1 0, E2 0, E3 0, E4 0} C_DIS
LIN {X 822.747, Y -10.817, Z 408, A 0, B 90, C -0, E1 0, E2 0, E3 0, E4 0} C_DIS
LIN {X 821.043, Y -12.2, Z 408, A 0, B 90, C -0, E1 0, E2 0, E3 0, E4 0} C_DIS
LIN {X 819.297, Y -13.528, Z 408, A 0, B 90, C -0, E1 0, E2 0, E3 0, E4 0} C_DIS
LIN {X 817.51, Y -14.802, Z 408, A 0, B 90, C -0, E1 0, E2 0, E3 0, E4 0} C_DIS
LIN {X 815.683, Y -16.018, Z 408, A 0, B 90, C -0, E1 0, E2 0, E3 0, E4 0} C_DIS
LIN {X 813.82, Y -17.176, Z 408, A 0, B 90, C -0, E1 0, E2 0, E3 0, E4 0} C_DIS
LIN {X 811.921, Y -18.276, Z 408, A 0, B 90, C -0, E1 0, E2 0, E3 0, E4 0} C_DIS
LIN {X 809.988, Y -19.315, Z 408, A 0, B 90, C -0, E1 0, E2 0, E3 0, E4 0} C_DIS
LIN {X 808.023, Y -20.293, Z 408, A 0, B 90, C -0, E1 0, E2 0, E3 0, E4 0} C_DIS
LIN {X 806.029, Y -21.209, Z 408, A 0, B 90, C -0, E1 0, E2 0, E3 0, E4 0} C_DIS
LIN {X 804.007, Y -22.061, Z 408, A 0, B 90, C -0, E1 0, E2 0, E3 0, E4 0} C_DIS
LIN {X 801.96, Y -22.85, Z 408, A 0, B 90, C -0, E1 0, E2 0, E3 0, E4 0} C_DIS
LIN {X 799.888, Y -23.574, Z 408, A 0, B 90, C -0, E1 0, E2 0, E3 0, E4 0} C_DIS
LIN {X 797.795, Y -24.232, Z 408, A 0, B 90, C -0, E1 0, E2 0, E3 0, E4 0} C_DIS
LIN {X 795.682, Y -24.825, Z 408, A 0, B 90, C -0, E1 0, E2 0, E3 0, E4 0} C_DIS
LIN {X 793.552, Y -25.351, Z 408, A 0, B 90, C -0, E1 0, E2 0, E3 0, E4 0} C_DIS
LIN {X 791.406, Y -25.81, Z 408, A 0, B 90, C -0, E1 0, E2 0, E3 0, E4 0} C_DIS
LIN {X 789.247, Y -26.201, Z 408, A 0, B 90, C -0, E1 0, E2 0, E3 0, E4 0} C_DIS
LIN {X 787.076, Y -26.524, Z 408, A 0, B 90, C -0, E1 0, E2 0, E3 0, E4 0} C_DIS
LIN {X 784.897, Y -26.778, Z 408, A 0, B 90, C -0, E1 0, E2 0, E3 0, E4 0} C_DIS
LIN {X 782.71, Y -26.964, Z 408, A 0, B 90, C -0, E1 0, E2 0, E3 0, E4 0} C_DIS
LIN {X 780.519, Y -27.082, Z 408, A 0, B 90, C -0, E1 0, E2 0, E3 0, E4 0} C_DIS
LIN {X 778.325, Y -27.13, Z 408, A 0, B 90, C -0, E1 0, E2 0, E3 0, E4 0} C_DIS
LIN {X 776.131, Y -27.11, Z 408, A 0, B 90, C -0, E1 0, E2 0, E3 0, E4 0} C_DIS
LIN {X 773.938, Y -27.02, Z 408, A 0, B 90, C -0, E1 0, E2 0, E3 0, E4 0} C_DIS
LIN {X 771.75, Y -26.862, Z 408, A 0, B 90, C -0, E1 0, E2 0, E3 0, E4 0} C_DIS
LIN {X 769.567, Y -26.635, Z 408, A 0, B 90, C -0, E1 0, E2 0, E3 0, E4 0} C_DIS
LIN {X 767.393, Y -26.34, Z 408, A 0, B 90, C -0, E1 0, E2 0, E3 0, E4 0} C_DIS
LIN {X 765.229, Y -25.976, Z 408, A 0, B 90, C -0, E1 0, E2 0, E3 0, E4 0} C_DIS
LIN {X 763.077, Y -25.545, Z 408, A 0, B 90, C -0, E1 0, E2 0, E3 0, E4 0} C_DIS
LIN {X 760.94, Y -25.046, Z 408, A 0, B 90, C -0, E1 0, E2 0, E3 0, E4 0} C_DIS
LIN {X 758.82, Y -24.481, Z 408, A 0, B 90, C -0, E1 0, E2 0, E3 0, E4 0} C_DIS
LIN {X 756.718, Y -23.849, Z 408, A 0, B 90, C -0, E1 0, E2 0, E3 0, E4 0} C_DIS
LIN {X 754.638, Y -23.151, Z 408, A 0, B 90, C -0, E1 0, E2 0, E3 0, E4 0} C_DIS
LIN {X 752.58, Y -22.389, Z 408, A 0, B 90, C -0, E1 0, E2 0, E3 0, E4 0} C_DIS
LIN {X 750.548, Y -21.562, Z 408, A 0, B 90, C -0, E1 0, E2 0, E3 0, E4 0} C_DIS
LIN {X 748.542, Y -20.672, Z 408, A 0, B 90, C -0, E1 0, E2 0, E3 0, E4 0} C_DIS
LIN {X 746.565, Y -19.719, Z 408, A 0, B 90, C -0, E1 0, E2 0, E3 0, E4 0} C_DIS
LIN {X 744.62, Y -18.705, Z 408, A 0, B 90, C -0, E1 0, E2 0, E3 0, E4 0} C_DIS
LIN {X 742.707, Y -17.63, Z 408, A 0, B 90, C -0, E1 0, E2 0, E3 0, E4 0} C_DIS
LIN {X 740.828, Y -16.495, Z 408, A 0, B 90, C -0, E1 0, E2 0, E3 0, E4 0} C_DIS
LIN {X 738.987, Y -15.302, Z 408, A 0, B 90, C -0, E1 0, E2 0, E3 0, E4 0} C_DIS
LIN {X 737.183, Y -14.052, Z 408, A 0, B 90, C -0, E1 0, E2 0, E3 0, E4 0} C_DIS
LIN {X 735.42, Y -12.745, Z 408, A 0, B 90, C -0, E1 0, E2 0, E3 0, E4 0} C_DIS
LIN {X 733.699, Y -11.384, Z 408, A 0, B 90, C -0, E1 0, E2 0, E3 0, E4 0} C_DIS
LIN {X 732.021, Y -9.97, Z 408, A 0, B 90, C -0, E1 0, E2 0, E3 0, E4 0} C_DIS
LIN {X 730.389, Y -8.503, Z 408, A 0, B 90, C -0, E1 0, E2 0, E3 0, E4 0} C_DIS
LIN {X 728.803, Y -6.986, Z 408, A 0, B 90, C -0, E1 0, E2 0, E3 0, E4 0} C_DIS
LIN {X 727.266, Y -5.42, Z 408, A 0, B 90, C -0, E1 0, E2 0, E3 0, E4 0} C_DIS
LIN {X 725.779, Y -3.807, Z 408, A 0, B 90, C -0, E1 0, E2 0, E3 0, E4 0} C_DIS
LIN {X 724.343, Y -2.147, Z 408, A 0, B 90, C -0, E1 0, E2 0, E3 0, E4 0} C_DIS
LIN {X 722.96, Y -0.443, Z 408, A 0, B 90, C -0, E1 0, E2 0, E3 0, E4 0} C_DIS
LIN {X 721.632, Y 1.303, Z 408, A 0, B 90, C -0, E1 0, E2 0, E3 0, E4 0} C_DIS
LIN {X 720.359, Y 3.09, Z 408, A 0, B 90, C -0, E1 0, E2 0, E3 0, E4 0} C_DIS
LIN {X 719.142, Y 4.917, Z 408, A 0, B 90, C -0, E1 0, E2 0, E3 0, E4 0} C_DIS
LIN {X 717.984, Y 6.78, Z 408, A 0, B 90, C -0, E1 0, E2 0, E3 0, E4 0} C_DIS
LIN {X 716.884, Y 8.679, Z 408, A 0, B 90, C -0, E1 0, E2 0, E3 0, E4 0} C_DIS
LIN {X 715.845, Y 10.612, Z 408, A 0, B 90, C -0, E1 0, E2 0, E3 0, E4 0} C_DIS
LIN {X 714.867, Y 12.576, Z 408, A 0, B 90, C -0, E1 0, E2 0, E3 0, E4 0} C_DIS
LIN {X 713.951, Y 14.571, Z 408, A 0, B 90, C -0, E1 0, E2 0, E3 0, E4 0} C_DIS
LIN {X 713.099, Y 16.593, Z 408, A 0, B 90, C -0, E1 0, E2 0, E3 0, E4 0} C_DIS
LIN {X 712.31, Y 18.64, Z 408, A 0, B 90, C -0, E1 0, E2 0, E3 0, E4 0} C_DIS
LIN {X 711.586, Y 20.712, Z 408, A 0, B 90, C -0, E1 0, E2 0, E3 0, E4 0} C_DIS
LIN {X 710.928, Y 22.805, Z 408, A 0, B 90, C -0, E1 0, E2 0, E3 0, E4 0} C_DIS
LIN {X 710.335, Y 24.918, Z 408, A 0, B 90, C -0, E1 0, E2 0, E3 0, E4 0} C_DIS
LIN {X 709.809, Y 27.048, Z 408, A 0, B 90, C -0, E1 0, E2 0, E3 0, E4 0} C_DIS
LIN {X 709.351, Y 29.194, Z 408, A 0, B 90, C -0, E1 0, E2 0, E3 0, E4 0} C_DIS
LIN {X 708.959, Y 31.353, Z 408, A 0, B 90, C -0, E1 0, E2 0, E3 0, E4 0} C_DIS
LIN {X 708.636, Y 33.524, Z 408, A 0, B 90, C -0, E1 0, E2 0, E3 0, E4 0} C_DIS
LIN {X 708.382, Y 35.703, Z 408, A 0, B 90, C -0, E1 0, E2 0, E3 0, E4 0} C_DIS
LIN {X 708.196, Y 37.89, Z 408, A 0, B 90, C -0, E1 0, E2 0, E3 0, E4 0} C_DIS
LIN {X 708.078, Y 40.081, Z 408, A 0, B 90, C -0, E1 0, E2 0, E3 0, E4 0} C_DIS
LIN {X 708.03, Y 42.275, Z 408, A 0, B 90, C -0, E1 0, E2 0, E3 0, E4 0} C_DIS
LIN {X 708.05, Y 44.469, Z 408, A 0, B 90, C -0, E1 0, E2 0, E3 0, E4 0} C_DIS
LIN {X 708.14, Y 46.662, Z 408, A 0, B 90, C -0, E1 0, E2 0, E3 0, E4 0} C_DIS
LIN {X 708.298, Y 48.85, Z 408, A 0, B 90, C -0, E1 0, E2 0, E3 0, E4 0} C_DIS
LIN {X 708.525, Y 51.033, Z 408, A 0, B 90, C -0, E1 0, E2 0, E3 0, E4 0} C_DIS
LIN {X 708.82, Y 53.207, Z 408, A 0, B 90, C -0, E1 0, E2 0, E3 0, E4 0} C_DIS
LIN {X 709.184, Y 55.371, Z 408, A 0, B 90, C -0, E1 0, E2 0, E3 0, E4 0} C_DIS
LIN {X 709.615, Y 57.523, Z 408, A 0, B 90, C -0, E1 0, E2 0, E3 0, E4 0} C_DIS
LIN {X 710.114, Y 59.66, Z 408, A 0, B 90, C -0, E1 0, E2 0, E3 0, E4 0} C_DIS
LIN {X 710.679, Y 61.78, Z 408, A 0, B 90, C -0, E1 0, E2 0, E3 0, E4 0} C_DIS
LIN {X 711.311, Y 63.882, Z 408, A 0, B 90, C -0, E1 0, E2 0, E3 0, E4 0} C_DIS
LIN {X 712.193, Y 65.311, Z 410, A 0, B 90, C -0, E1 0, E2 0, E3 0, E4 0} C_DIS
LIN {X 712.935, Y 67.363, Z 410, A 0, B 90, C -0, E1 0, E2 0, E3 0, E4 0} C_DIS
LIN {X 713.741, Y 69.391, Z 410, A 0, B 90, C -0, E1 0, E2 0, E3 0, E4 0} C_DIS
LIN {X 714.61, Y 71.392, Z 410, A 0, B 90, C -0, E1 0, E2 0, E3 0, E4 0} C_DIS
LIN {X 715.542, Y 73.366, Z 410, A 0, B 90, C -0, E1 0, E2 0, E3 0, E4 0} C_DIS
LIN {X 716.536, Y 75.309, Z 410, A 0, B 90, C -0, E1 0, E2 0, E3 0, E4 0} C_DIS
LIN {X 717.59, Y 77.219, Z 410, A 0, B 90, C -0, E1 0, E2 0, E3 0, E4 0} C_DIS
LIN {X 718.703, Y 79.096, Z 410, A 0, B 90, C -0, E1 0, E2 0, E3 0, E4 0} C_DIS
LIN {X 719.875, Y 80.937, Z 410, A 0, B 90, C -0, E1 0, E2 0, E3 0, E4 0} C_DIS
LIN {X 721.104, Y 82.74, Z 410, A 0, B 90, C -0, E1 0, E2 0, E3 0, E4 0} C_DIS
LIN {X 722.389, Y 84.504, Z 410, A 0, B 90, C -0, E1 0, E2 0, E3 0, E4 0} C_DIS
LIN {X 723.729, Y 86.226, Z 410, A 0, B 90, C -0, E1 0, E2 0, E3 0, E4 0} C_DIS
LIN {X 725.122, Y 87.906, Z 410, A 0, B 90, C -0, E1 0, E2 0, E3 0, E4 0} C_DIS
LIN {X 726.567, Y 89.54, Z 410, A 0, B 90, C -0, E1 0, E2 0, E3 0, E4 0} C_DIS
LIN {X 728.063, Y 91.129, Z 410, A 0, B 90, C -0, E1 0, E2 0, E3 0, E4 0} C_DIS
LIN {X 729.608, Y 92.67, Z 410, A 0, B 90, C -0, E1 0, E2 0, E3 0, E4 0} C_DIS
LIN {X 731.201, Y 94.162, Z 410, A 0, B 90, C -0, E1 0, E2 0, E3 0, E4 0} C_DIS
LIN {X 732.84, Y 95.602, Z 410, A 0, B 90, C -0, E1 0, E2 0, E3 0, E4 0} C_DIS
LIN {X 734.523, Y 96.991, Z 410, A 0, B 90, C -0, E1 0, E2 0, E3 0, E4 0} C_DIS
LIN {X 736.25, Y 98.326, Z 410, A 0, B 90, C -0, E1 0, E2 0, E3 0, E4 0} C_DIS
LIN {X 738.017, Y 99.606, Z 410, A 0, B 90, C -0, E1 0, E2 0, E3 0, E4 0} C_DIS
LIN {X 739.823, Y 100.83, Z 410, A 0, B 90, C -0, E1 0, E2 0, E3 0, E4 0} C_DIS
LIN {X 741.667, Y 101.997, Z 410, A 0, B 90, C -0, E1 0, E2 0, E3 0, E4 0} C_DIS
LIN {X 743.547, Y 103.105, Z 410, A 0, B 90, C -0, E1 0, E2 0, E3 0, E4 0} C_DIS
LIN {X 745.461, Y 104.154, Z 410, A 0, B 90, C -0, E1 0, E2 0, E3 0, E4 0} C_DIS
LIN {X 747.406, Y 105.142, Z 410, A 0, B 90, C -0, E1 0, E2 0, E3 0, E4 0} C_DIS
LIN {X 749.382, Y 106.068, Z 410, A 0, B 90, C -0, E1 0, E2 0, E3 0, E4 0} C_DIS
LIN {X 751.386, Y 106.932, Z 410, A 0, B 90, C -0, E1 0, E2 0, E3 0, E4 0} C_DIS
LIN {X 753.416, Y 107.733, Z 410, A 0, B 90, C -0, E1 0, E2 0, E3 0, E4 0} C_DIS
LIN {X 755.47, Y 108.469, Z 410, A 0, B 90, C -0, E1 0, E2 0, E3 0, E4 0} C_DIS
LIN {X 757.547, Y 109.141, Z 410, A 0, B 90, C -0, E1 0, E2 0, E3 0, E4 0} C_DIS
LIN {X 759.643, Y 109.747, Z 410, A 0, B 90, C -0, E1 0, E2 0, E3 0, E4 0} C_DIS
LIN {X 761.757, Y 110.286, Z 410, A 0, B 90, C -0, E1 0, E2 0, E3 0, E4 0} C_DIS
LIN {X 763.888, Y 110.759, Z 410, A 0, B 90, C -0, E1 0, E2 0, E3 0, E4 0} C_DIS
LIN {X 766.032, Y 111.165, Z 410, A 0, B 90, C -0, E1 0, E2 0, E3 0, E4 0} C_DIS
LIN {X 768.187, Y 111.504, Z 410, A 0, B 90, C -0, E1 0, E2 0, E3 0, E4 0} C_DIS
LIN {X 770.353, Y 111.774, Z 410, A 0, B 90, C -0, E1 0, E2 0, E3 0, E4 0} C_DIS
LIN {X 772.526, Y 111.977, Z 410, A 0, B 90, C -0, E1 0, E2 0, E3 0, E4 0} C_DIS
LIN {X 774.704, Y 112.111, Z 410, A 0, B 90, C -0, E1 0, E2 0, E3 0, E4 0} C_DIS
LIN {X 776.885, Y 112.176, Z 410, A 0, B 90, C -0, E1 0, E2 0, E3 0, E4 0} C_DIS
LIN {X 779.067, Y 112.173, Z 410, A 0, B 90, C -0, E1 0, E2 0, E3 0, E4 0} C_DIS
LIN {X 781.248, Y 112.102, Z 410, A 0, B 90, C -0, E1 0, E2 0, E3 0, E4 0} C_DIS
LIN {X 783.426, Y 111.962, Z 410, A 0, B 90, C -0, E1 0, E2 0, E3 0, E4 0} C_DIS
LIN {X 785.598, Y 111.753, Z 410, A 0, B 90, C -0, E1 0, E2 0, E3 0, E4 0} C_DIS
LIN {X 787.762, Y 111.477, Z 410, A 0, B 90, C -0, E1 0, E2 0, E3 0, E4 0} C_DIS
LIN {X 789.917, Y 111.132, Z 410, A 0, B 90, C -0, E1 0, E2 0, E3 0, E4 0} C_DIS
LIN {X 792.06, Y 110.721, Z 410, A 0, B 90, C -0, E1 0, E2 0, E3 0, E4 0} C_DIS
LIN {X 794.189, Y 110.242, Z 410, A 0, B 90, C -0, E1 0, E2 0, E3 0, E4 0} C_DIS
LIN {X 796.302, Y 109.696, Z 410, A 0, B 90, C -0, E1 0, E2 0, E3 0, E4 0} C_DIS
LIN {X 798.397, Y 109.084, Z 410, A 0, B 90, C -0, E1 0, E2 0, E3 0, E4 0} C_DIS
LIN {X 800.471, Y 108.407, Z 410, A 0, B 90, C -0, E1 0, E2 0, E3 0, E4 0} C_DIS
LIN {X 802.523, Y 107.665, Z 410, A 0, B 90, C -0, E1 0, E2 0, E3 0, E4 0} C_DIS
LIN {X 804.551, Y 106.859, Z 410, A 0, B 90, C -0, E1 0, E2 0, E3 0, E4 0} C_DIS
LIN {X 806.552, Y 105.99, Z 410, A 0, B 90, C -0, E1 0, E2 0, E3 0, E4 0} C_DIS
LIN {X 808.526, Y 105.058, Z 410, A 0, B 90, C -0, E1 0, E2 0, E3 0, E4 0} C_DIS
LIN {X 810.469, Y 104.064, Z 410, A 0, B 90, C -0, E1 0, E2 0, E3 0, E4 0} C_DIS
LIN {X 812.379, Y 103.01, Z 410, A 0, B 90, C -0, E1 0, E2 0, E3 0, E4 0} C_DIS
LIN {X 814.256, Y 101.897, Z 410, A 0, B 90, C -0, E1 0, E2 0, E3 0, E4 0} C_DIS
LIN {X 816.097, Y 100.725, Z 410, A 0, B 90, C -0, E1 0, E2 0, E3 0, E4 0} C_DIS
LIN {X 817.9, Y 99.496, Z 410, A 0, B 90, C -0, E1 0, E2 0, E3 0, E4 0} C_DIS
LIN {X 819.664, Y 98.211, Z 410, A 0, B 90, C -0, E1 0, E2 0, E3 0, E4 0} C_DIS
LIN {X 821.386, Y 96.871, Z 410, A 0, B 90, C -0, E1 0, E2 0, E3 0, E4 0} C_DIS
LIN {X 823.066, Y 95.478, Z 410, A 0, B 90, C -0, E1 0, E2 0, E3 0, E4 0} C_DIS
LIN {X 824.701, Y 94.033, Z 410, A 0, B 90, C -0, E1 0, E2 0, E3 0, E4 0} C_DIS
LIN {X 826.289, Y 92.537, Z 410, A 0, B 90, C -0, E1 0, E2 0, E3 0, E4 0} C_DIS
LIN {X 827.83, Y 90.992, Z 410, A 0, B 90, C -0, E1 0, E2 0, E3 0, E4 0} C_DIS
LIN {X 829.322, Y 89.399, Z 410, A 0, B 90, C -0, E1 0, E2 0, E3 0, E4 0} C_DIS
LIN {X 830.762, Y 87.76, Z 410, A 0, B 90, C -0, E1 0, E2 0, E3 0, E4 0} C_DIS
LIN {X 832.151, Y 86.077, Z 410, A 0, B 90, C -0, E1 0, E2 0, E3 0, E4 0} C_DIS
LIN {X 833.486, Y 84.35, Z 410, A 0, B 90, C -0, E1 0, E2 0, E3 0, E4 0} C_DIS
LIN {X 834.766, Y 82.583, Z 410, A 0, B 90, C -0, E1 0, E2 0, E3 0, E4 0} C_DIS
LIN {X 835.99, Y 80.777, Z 410, A 0, B 90, C -0, E1 0, E2 0, E3 0, E4 0} C_DIS
LIN {X 837.157, Y 78.933, Z 410, A 0, B 90, C -0, E1 0, E2 0, E3 0, E4 0} C_DIS
LIN {X 838.265, Y 77.053, Z 410, A 0, B 90, C -0, E1 0, E2 0, E3 0, E4 0} C_DIS
LIN {X 839.314, Y 75.139, Z 410, A 0, B 90, C -0, E1 0, E2 0, E3 0, E4 0} C_DIS
LIN {X 840.302, Y 73.194, Z 410, A 0, B 90, C -0, E1 0, E2 0, E3 0, E4 0} C_DIS
LIN {X 841.228, Y 71.218, Z 410, A 0, B 90, C -0, E1 0, E2 0, E3 0, E4 0} C_DIS
LIN {X 842.092, Y 69.214, Z 410, A 0, B 90, C -0, E1 0, E2 0, E3 0, E4 0} C_DIS
LIN {X 842.893, Y 67.184, Z 410, A 0, B 90, C -0, E1 0, E2 0, E3 0, E4 0} C_DIS
LIN {X 843.629, Y 65.13, Z 410, A 0, B 90, C -0, E1 0, E2 0, E3 0, E4 0} C_DIS
LIN {X 844.301, Y 63.053, Z 410, A 0, B 90, C -0, E1 0, E2 0, E3 0, E4 0} C_DIS
LIN {X 844.907, Y 60.957, Z 410, A 0, B 90, C -0, E1 0, E2 0, E3 0, E4 0} C_DIS
LIN {X 845.446, Y 58.843, Z 410, A 0, B 90, C -0, E1 0, E2 0, E3 0, E4 0} C_DIS
LIN {X 845.919, Y 56.712, Z 410, A 0, B 90, C -0, E1 0, E2 0, E3 0, E4 0} C_DIS
LIN {X 846.325, Y 54.568, Z 410, A 0, B 90, C -0, E1 0, E2 0, E3 0, E4 0} C_DIS
LIN {X 846.664, Y 52.413, Z 410, A 0, B 90, C -0, E1 0, E2 0, E3 0, E4 0} C_DIS
LIN {X 846.934, Y 50.247, Z 410, A 0, B 90, C -0, E1 0, E2 0, E3 0, E4 0} C_DIS
LIN {X 847.137, Y 48.074, Z 410, A 0, B 90, C -0, E1 0, E2 0, E3 0, E4 0} C_DIS
LIN {X 847.271, Y 45.896, Z 410, A 0, B 90, C -0, E1 0, E2 0, E3 0, E4 0} C_DIS
LIN {X 847.336, Y 43.715, Z 410, A 0, B 90, C -0, E1 0, E2 0, E3 0, E4 0} C_DIS
LIN {X 847.333, Y 41.533, Z 410, A 0, B 90, C -0, E1 0, E2 0, E3 0, E4 0} C_DIS
LIN {X 847.262, Y 39.352, Z 410, A 0, B 90, C -0, E1 0, E2 0, E3 0, E4 0} C_DIS
LIN {X 847.122, Y 37.174, Z 410, A 0, B 90, C -0, E1 0, E2 0, E3 0, E4 0} C_DIS
LIN {X 846.913, Y 35.002, Z 410, A 0, B 90, C -0, E1 0, E2 0, E3 0, E4 0} C_DIS
LIN {X 846.637, Y 32.838, Z 410, A 0, B 90, C -0, E1 0, E2 0, E3 0, E4 0} C_DIS
LIN {X 846.292, Y 30.683, Z 410, A 0, B 90, C -0, E1 0, E2 0, E3 0, E4 0} C_DIS
LIN {X 845.88, Y 28.54, Z 410, A 0, B 90, C -0, E1 0, E2 0, E3 0, E4 0} C_DIS
LIN {X 845.402, Y 26.411, Z 410, A 0, B 90, C -0, E1 0, E2 0, E3 0, E4 0} C_DIS
LIN {X 844.856, Y 24.298, Z 410, A 0, B 90, C -0, E1 0, E2 0, E3 0, E4 0} C_DIS
LIN {X 844.244, Y 22.203, Z 410, A 0, B 90, C -0, E1 0, E2 0, E3 0, E4 0} C_DIS
LIN {X 843.567, Y 20.129, Z 410, A 0, B 90, C -0, E1 0, E2 0, E3 0, E4 0} C_DIS
LIN {X 842.825, Y 18.077, Z 410, A 0, B 90, C -0, E1 0, E2 0, E3 0, E4 0} C_DIS
LIN {X 842.019, Y 16.049, Z 410, A 0, B 90, C -0, E1 0, E2 0, E3 0, E4 0} C_DIS
LIN {X 841.15, Y 14.048, Z 410, A 0, B 90, C -0, E1 0, E2 0, E3 0, E4 0} C_DIS
LIN {X 840.218, Y 12.074, Z 410, A 0, B 90, C -0, E1 0, E2 0, E3 0, E4 0} C_DIS
LIN {X 839.224, Y 10.131, Z 410, A 0, B 90, C -0, E1 0, E2 0, E3 0, E4 0} C_DIS
LIN {X 838.17, Y 8.221, Z 410, A 0, B 90, C -0, E1 0, E2 0, E3 0, E4 0} C_DIS
LIN {X 837.057, Y 6.344, Z 410, A 0, B 90, C -0, E1 0, E2 0, E3 0, E4 0} C_DIS
LIN {X 835.885, Y 4.503, Z 410, A 0, B 90, C -0, E1 0, E2 0, E3 0, E4 0} C_DIS
LIN {X 834.656, Y 2.7, Z 410, A 0, B 90, C -0, E1 0, E2 0, E3 0, E4 0} C_DIS
LIN {X 833.371, Y 0.936, Z 410, A 0, B 90, C -0, E1 0, E2 0, E3 0, E4 0} C_DIS
LIN {X 832.031, Y -0.786, Z 410, A 0, B 90, C -0, E1 0, E2 0, E3 0, E4 0} C_DIS
LIN {X 830.638, Y -2.466, Z 410, A 0, B 90, C -0, E1 0, E2 0, E3 0, E4 0} C_DIS
LIN {X 829.193, Y -4.1, Z 410, A 0, B 90, C -0, E1 0, E2 0, E3 0, E4 0} C_DIS
LIN {X 827.697, Y -5.689, Z 410, A 0, B 90, C -0, E1 0, E2 0, E3 0, E4 0} C_DIS
LIN {X 826.151, Y -7.23, Z 410, A 0, B 90, C -0, E1 0, E2 0, E3 0, E4 0} C_DIS
LIN {X 824.559, Y -8.722, Z 410, A 0, B 90, C -0, E1 0, E2 0, E3 0, E4 0} C_DIS
LIN {X 822.92, Y -10.162, Z 410, A 0, B 90, C -0, E1 0, E2 0, E3 0, E4 0} C_DIS
LIN {X 821.237, Y -11.551, Z 410, A 0, B 90, C -0, E1 0, E2 0, E3 0, E4 0} C_DIS
LIN {X 819.51, Y -12.886, Z 410, A 0, B 90, C -0, E1 0, E2 0, E3 0, E4 0} C_DIS
LIN {X 817.743, Y -14.166, Z 410, A 0, B 90, C -0, E1 0, E2 0, E3 0, E4 0} C_DIS
LIN {X 815.937, Y -15.39, Z 410, A 0, B 90, C -0, E1 0, E2 0, E3 0, E4 0} C_DIS
LIN {X 814.093, Y -16.557, Z 410, A 0, B 90, C -0, E1 0, E2 0, E3 0, E4 0} C_DIS
LIN {X 812.213, Y -17.665, Z 410, A 0, B 90, C -0, E1 0, E2 0, E3 0, E4 0} C_DIS
LIN {X 810.299, Y -18.714, Z 410, A 0, B 90, C -0, E1 0, E2 0, E3 0, E4 0} C_DIS
LIN {X 808.354, Y -19.702, Z 410, A 0, B 90, C -0, E1 0, E2 0, E3 0, E4 0} C_DIS
LIN {X 806.378, Y -20.628, Z 410, A 0, B 90, C -0, E1 0, E2 0, E3 0, E4 0} C_DIS
LIN {X 804.374, Y -21.492, Z 410, A 0, B 90, C -0, E1 0, E2 0, E3 0, E4 0} C_DIS
LIN {X 802.344, Y -22.293, Z 410, A 0, B 90, C -0, E1 0, E2 0, E3 0, E4 0} C_DIS
LIN {X 800.29, Y -23.029, Z 410, A 0, B 90, C -0, E1 0, E2 0, E3 0, E4 0} C_DIS
LIN {X 798.213, Y -23.701, Z 410, A 0, B 90, C -0, E1 0, E2 0, E3 0, E4 0} C_DIS
LIN {X 796.117, Y -24.307, Z 410, A 0, B 90, C -0, E1 0, E2 0, E3 0, E4 0} C_DIS
LIN {X 794.003, Y -24.846, Z 410, A 0, B 90, C -0, E1 0, E2 0, E3 0, E4 0} C_DIS
LIN {X 791.872, Y -25.319, Z 410, A 0, B 90, C -0, E1 0, E2 0, E3 0, E4 0} C_DIS
LIN {X 789.728, Y -25.725, Z 410, A 0, B 90, C -0, E1 0, E2 0, E3 0, E4 0} C_DIS
LIN {X 787.573, Y -26.064, Z 410, A 0, B 90, C -0, E1 0, E2 0, E3 0, E4 0} C_DIS
LIN {X 785.407, Y -26.334, Z 410, A 0, B 90, C -0, E1 0, E2 0, E3 0, E4 0} C_DIS
LIN {X 783.234, Y -26.537, Z 410, A 0, B 90, C -0, E1 0, E2 0, E3 0, E4 0} C_DIS
LIN {X 781.056, Y -26.671, Z 410, A 0, B 90, C -0, E1 0, E2 0, E3 0, E4 0} C_DIS
LIN {X 778.875, Y -26.736, Z 410, A 0, B 90, C -0, E1 0, E2 0, E3 0, E4 0} C_DIS
LIN {X 776.693, Y -26.733, Z 410, A 0, B 90, C -0, E1 0, E2 0, E3 0, E4 0} C_DIS
LIN {X 774.512, Y -26.662, Z 410, A 0, B 90, C -0, E1 0, E2 0, E3 0, E4 0} C_DIS
LIN {X 772.334, Y -26.522, Z 410, A 0, B 90, C -0, E1 0, E2 0, E3 0, E4 0} C_DIS
LIN {X 770.162, Y -26.313, Z 410, A 0, B 90, C -0, E1 0, E2 0, E3 0, E4 0} C_DIS
LIN {X 767.998, Y -26.037, Z 410, A 0, B 90, C -0, E1 0, E2 0, E3 0, E4 0} C_DIS
LIN {X 765.843, Y -25.692, Z 410, A 0, B 90, C -0, E1 0, E2 0, E3 0, E4 0} C_DIS
LIN {X 763.7, Y -25.281, Z 410, A 0, B 90, C -0, E1 0, E2 0, E3 0, E4 0} C_DIS
LIN {X 761.571, Y -24.802, Z 410, A 0, B 90, C -0, E1 0, E2 0, E3 0, E4 0} C_DIS
LIN {X 759.458, Y -24.256, Z 410, A 0, B 90, C -0, E1 0, E2 0, E3 0, E4 0} C_DIS
LIN {X 757.363, Y -23.644, Z 410, A 0, B 90, C -0, E1 0, E2 0, E3 0, E4 0} C_DIS
LIN {X 755.289, Y -22.967, Z 410, A 0, B 90, C -0, E1 0, E2 0, E3 0, E4 0} C_DIS
LIN {X 753.237, Y -22.225, Z 410, A 0, B 90, C -0, E1 0, E2 0, E3 0, E4 0} C_DIS
LIN {X 751.209, Y -21.419, Z 410, A 0, B 90, C -0, E1 0, E2 0, E3 0, E4 0} C_DIS
LIN {X 749.208, Y -20.55, Z 410, A 0, B 90, C -0, E1 0, E2 0, E3 0, E4 0} C_DIS
LIN {X 747.234, Y -19.618, Z 410, A 0, B 90, C -0, E1 0, E2 0, E3 0, E4 0} C_DIS
LIN {X 745.291, Y -18.624, Z 410, A 0, B 90, C -0, E1 0, E2 0, E3 0, E4 0} C_DIS
LIN {X 743.381, Y -17.57, Z 410, A 0, B 90, C -0, E1 0, E2 0, E3 0, E4 0} C_DIS
LIN {X 741.504, Y -16.457, Z 410, A 0, B 90, C -0, E1 0, E2 0, E3 0, E4 0} C_DIS
LIN {X 739.663, Y -15.285, Z 410, A 0, B 90, C -0, E1 0, E2 0, E3 0, E4 0} C_DIS
LIN {X 737.86, Y -14.056, Z 410, A 0, B 90, C -0, E1 0, E2 0, E3 0, E4 0} C_DIS
LIN {X 736.096, Y -12.771, Z 410, A 0, B 90, C -0, E1 0, E2 0, E3 0, E4 0} C_DIS
LIN {X 734.374, Y -11.431, Z 410, A 0, B 90, C -0, E1 0, E2 0, E3 0, E4 0} C_DIS
LIN {X 732.694, Y -10.038, Z 410, A 0, B 90, C -0, E1 0, E2 0, E3 0, E4 0} C_DIS
LIN {X 731.06, Y -8.593, Z 410, A 0, B 90, C -0, E1 0, E2 0, E3 0, E4 0} C_DIS
LIN {X 729.471, Y -7.097, Z 410, A 0, B 90, C -0, E1 0, E2 0, E3 0, E4 0} C_DIS
LIN {X 727.93, Y -5.552, Z 410, A 0, B 90, C -0, E1 0, E2 0, E3 0, E4 0} C_DIS
LIN {X 726.438, Y -3.959, Z 410, A 0, B 90, C -0, E1 0, E2 0, E3 0, E4 0} C_DIS
LIN {X 724.998, Y -2.32, Z 410, A 0, B 90, C -0, E1 0, E2 0, E3 0, E4 0} C_DIS
LIN {X 723.609, Y -0.637, Z 410, A 0, B 90, C -0, E1 0, E2 0, E3 0, E4 0} C_DIS
LIN {X 722.274, Y 1.09, Z 410, A 0, B 90, C -0, E1 0, E2 0, E3 0, E4 0} C_DIS
LIN {X 720.994, Y 2.857, Z 410, A 0, B 90, C -0, E1 0, E2 0, E3 0, E4 0} C_DIS
LIN {X 719.77, Y 4.663, Z 410, A 0, B 90, C -0, E1 0, E2 0, E3 0, E4 0} C_DIS
LIN {X 718.603, Y 6.507, Z 410, A 0, B 90, C -0, E1 0, E2 0, E3 0, E4 0} C_DIS
LIN {X 717.495, Y 8.387, Z 410, A 0, B 90, C -0, E1 0, E2 0, E3 0, E4 0} C_DIS
LIN {X 716.446, Y 10.301, Z 410, A 0, B 90, C -0, E1 0, E2 0, E3 0, E4 0} C_DIS
LIN {X 715.458, Y 12.246, Z 410, A 0, B 90, C -0, E1 0, E2 0, E3 0, E4 0} C_DIS
LIN {X 714.532, Y 14.222, Z 410, A 0, B 90, C -0, E1 0, E2 0, E3 0, E4 0} C_DIS
LIN {X 713.668, Y 16.226, Z 410, A 0, B 90, C -0, E1 0, E2 0, E3 0, E4 0} C_DIS
LIN {X 712.867, Y 18.256, Z 410, A 0, B 90, C -0, E1 0, E2 0, E3 0, E4 0} C_DIS
LIN {X 712.131, Y 20.31, Z 410, A 0, B 90, C -0, E1 0, E2 0, E3 0, E4 0} C_DIS
LIN {X 711.459, Y 22.387, Z 410, A 0, B 90, C -0, E1 0, E2 0, E3 0, E4 0} C_DIS
LIN {X 710.853, Y 24.483, Z 410, A 0, B 90, C -0, E1 0, E2 0, E3 0, E4 0} C_DIS
LIN {X 710.314, Y 26.597, Z 410, A 0, B 90, C -0, E1 0, E2 0, E3 0, E4 0} C_DIS
LIN {X 709.841, Y 28.728, Z 410, A 0, B 90, C -0, E1 0, E2 0, E3 0, E4 0} C_DIS
LIN {X 709.435, Y 30.872, Z 410, A 0, B 90, C -0, E1 0, E2 0, E3 0, E4 0} C_DIS
LIN {X 709.096, Y 33.027, Z 410, A 0, B 90, C -0, E1 0, E2 0, E3 0, E4 0} C_DIS
LIN {X 708.826, Y 35.193, Z 410, A 0, B 90, C -0, E1 0, E2 0, E3 0, E4 0} C_DIS
LIN {X 708.623, Y 37.366, Z 410, A 0, B 90, C -0, E1 0, E2 0, E3 0, E4 0} C_DIS
LIN {X 708.489, Y 39.544, Z 410, A 0, B 90, C -0, E1 0, E2 0, E3 0, E4 0} C_DIS
LIN {X 708.424, Y 41.725, Z 410, A 0, B 90, C -0, E1 0, E2 0, E3 0, E4 0} C_DIS
LIN {X 708.427, Y 43.907, Z 410, A 0, B 90, C -0, E1 0, E2 0, E3 0, E4 0} C_DIS
LIN {X 708.498, Y 46.088, Z 410, A 0, B 90, C -0, E1 0, E2 0, E3 0, E4 0} C_DIS
LIN {X 708.638, Y 48.266, Z 410, A 0, B 90, C -0, E1 0, E2 0, E3 0, E4 0} C_DIS
LIN {X 708.847, Y 50.438, Z 410, A 0, B 90, C -0, E1 0, E2 0, E3 0, E4 0} C_DIS
LIN {X 709.123, Y 52.602, Z 410, A 0, B 90, C -0, E1 0, E2 0, E3 0, E4 0} C_DIS
LIN {X 709.468, Y 54.757, Z 410, A 0, B 90, C -0, E1 0, E2 0, E3 0, E4 0} C_DIS
LIN {X 709.879, Y 56.9, Z 410, A 0, B 90, C -0, E1 0, E2 0, E3 0, E4 0} C_DIS
LIN {X 710.358, Y 59.029, Z 410, A 0, B 90, C -0, E1 0, E2 0, E3 0, E4 0} C_DIS
LIN {X 710.904, Y 61.142, Z 410, A 0, B 90, C -0, E1 0, E2 0, E3 0, E4 0} C_DIS
LIN {X 711.516, Y 63.237, Z 410, A 0, B 90, C -0, E1 0, E2 0, E3 0, E4 0} C_DIS
LIN {X 712.381, Y 64.676, Z 412, A 0, B 90, C -0, E1 0, E2 0, E3 0, E4 0} C_DIS
LIN {X 713.103, Y 66.723, Z 412, A 0, B 90, C -0, E1 0, E2 0, E3 0, E4 0} C_DIS
LIN {X 713.889, Y 68.746, Z 412, A 0, B 90, C -0, E1 0, E2 0, E3 0, E4 0} C_DIS
LIN {X 714.738, Y 70.743, Z 412, A 0, B 90, C -0, E1 0, E2 0, E3 0, E4 0} C_DIS
LIN {X 715.649, Y 72.712, Z 412, A 0, B 90, C -0, E1 0, E2 0, E3 0, E4 0} C_DIS
LIN {X 716.622, Y 74.652, Z 412, A 0, B 90, C -0, E1 0, E2 0, E3 0, E4 0} C_DIS
LIN {X 717.655, Y 76.561, Z 412, A 0, B 90, C -0, E1 0, E2 0, E3 0, E4 0} C_DIS
LIN {X 718.748, Y 78.436, Z 412, A 0, B 90, C -0, E1 0, E2 0, E3 0, E4 0} C_DIS
LIN {X 719.899, Y 80.275, Z 412, A 0, B 90, C -0, E1 0, E2 0, E3 0, E4 0} C_DIS
LIN {X 721.107, Y 82.078, Z 412, A 0, B 90, C -0, E1 0, E2 0, E3 0, E4 0} C_DIS
LIN {X 722.371, Y 83.842, Z 412, A 0, B 90, C -0, E1 0, E2 0, E3 0, E4 0} C_DIS
LIN {X 723.69, Y 85.565, Z 412, A 0, B 90, C -0, E1 0, E2 0, E3 0, E4 0} C_DIS
LIN {X 725.063, Y 87.246, Z 412, A 0, B 90, C -0, E1 0, E2 0, E3 0, E4 0} C_DIS
LIN {X 726.487, Y 88.883, Z 412, A 0, B 90, C -0, E1 0, E2 0, E3 0, E4 0} C_DIS
LIN {X 727.963, Y 90.475, Z 412, A 0, B 90, C -0, E1 0, E2 0, E3 0, E4 0} C_DIS
LIN {X 729.488, Y 92.019, Z 412, A 0, B 90, C -0, E1 0, E2 0, E3 0, E4 0} C_DIS
LIN {X 731.06, Y 93.515, Z 412, A 0, B 90, C -0, E1 0, E2 0, E3 0, E4 0} C_DIS
LIN {X 732.679, Y 94.961, Z 412, A 0, B 90, C -0, E1 0, E2 0, E3 0, E4 0} C_DIS
LIN {X 734.342, Y 96.355, Z 412, A 0, B 90, C -0, E1 0, E2 0, E3 0, E4 0} C_DIS
LIN {X 736.048, Y 97.696, Z 412, A 0, B 90, C -0, E1 0, E2 0, E3 0, E4 0} C_DIS
LIN {X 737.795, Y 98.983, Z 412, A 0, B 90, C -0, E1 0, E2 0, E3 0, E4 0} C_DIS
LIN {X 739.582, Y 100.214, Z 412, A 0, B 90, C -0, E1 0, E2 0, E3 0, E4 0} C_DIS
LIN {X 741.407, Y 101.388, Z 412, A 0, B 90, C -0, E1 0, E2 0, E3 0, E4 0} C_DIS
LIN {X 743.268, Y 102.505, Z 412, A 0, B 90, C -0, E1 0, E2 0, E3 0, E4 0} C_DIS
LIN {X 745.163, Y 103.563, Z 412, A 0, B 90, C -0, E1 0, E2 0, E3 0, E4 0} C_DIS
LIN {X 747.09, Y 104.56, Z 412, A 0, B 90, C -0, E1 0, E2 0, E3 0, E4 0} C_DIS
LIN {X 749.048, Y 105.497, Z 412, A 0, B 90, C -0, E1 0, E2 0, E3 0, E4 0} C_DIS
LIN {X 751.034, Y 106.372, Z 412, A 0, B 90, C -0, E1 0, E2 0, E3 0, E4 0} C_DIS
LIN {X 753.047, Y 107.184, Z 412, A 0, B 90, C -0, E1 0, E2 0, E3 0, E4 0} C_DIS
LIN {X 755.084, Y 107.932, Z 412, A 0, B 90, C -0, E1 0, E2 0, E3 0, E4 0} C_DIS
LIN {X 757.143, Y 108.616, Z 412, A 0, B 90, C -0, E1 0, E2 0, E3 0, E4 0} C_DIS
LIN {X 759.223, Y 109.234, Z 412, A 0, B 90, C -0, E1 0, E2 0, E3 0, E4 0} C_DIS
LIN {X 761.322, Y 109.788, Z 412, A 0, B 90, C -0, E1 0, E2 0, E3 0, E4 0} C_DIS
LIN {X 763.437, Y 110.275, Z 412, A 0, B 90, C -0, E1 0, E2 0, E3 0, E4 0} C_DIS
LIN {X 765.566, Y 110.695, Z 412, A 0, B 90, C -0, E1 0, E2 0, E3 0, E4 0} C_DIS
LIN {X 767.707, Y 111.048, Z 412, A 0, B 90, C -0, E1 0, E2 0, E3 0, E4 0} C_DIS
LIN {X 769.858, Y 111.334, Z 412, A 0, B 90, C -0, E1 0, E2 0, E3 0, E4 0} C_DIS
LIN {X 772.017, Y 111.552, Z 412, A 0, B 90, C -0, E1 0, E2 0, E3 0, E4 0} C_DIS
LIN {X 774.182, Y 111.702, Z 412, A 0, B 90, C -0, E1 0, E2 0, E3 0, E4 0} C_DIS
LIN {X 776.351, Y 111.784, Z 412, A 0, B 90, C -0, E1 0, E2 0, E3 0, E4 0} C_DIS
LIN {X 778.521, Y 111.798, Z 412, A 0, B 90, C -0, E1 0, E2 0, E3 0, E4 0} C_DIS
LIN {X 780.691, Y 111.744, Z 412, A 0, B 90, C -0, E1 0, E2 0, E3 0, E4 0} C_DIS
LIN {X 782.857, Y 111.622, Z 412, A 0, B 90, C -0, E1 0, E2 0, E3 0, E4 0} C_DIS
LIN {X 785.019, Y 111.432, Z 412, A 0, B 90, C -0, E1 0, E2 0, E3 0, E4 0} C_DIS
LIN {X 787.174, Y 111.173, Z 412, A 0, B 90, C -0, E1 0, E2 0, E3 0, E4 0} C_DIS
LIN {X 789.32, Y 110.848, Z 412, A 0, B 90, C -0, E1 0, E2 0, E3 0, E4 0} C_DIS
LIN {X 791.454, Y 110.455, Z 412, A 0, B 90, C -0, E1 0, E2 0, E3 0, E4 0} C_DIS
LIN {X 793.575, Y 109.995, Z 412, A 0, B 90, C -0, E1 0, E2 0, E3 0, E4 0} C_DIS
LIN {X 795.68, Y 109.469, Z 412, A 0, B 90, C -0, E1 0, E2 0, E3 0, E4 0} C_DIS
LIN {X 797.768, Y 108.877, Z 412, A 0, B 90, C -0, E1 0, E2 0, E3 0, E4 0} C_DIS
LIN {X 799.836, Y 108.219, Z 412, A 0, B 90, C -0, E1 0, E2 0, E3 0, E4 0} C_DIS
LIN {X 801.883, Y 107.497, Z 412, A 0, B 90, C -0, E1 0, E2 0, E3 0, E4 0} C_DIS
LIN {X 803.906, Y 106.711, Z 412, A 0, B 90, C -0, E1 0, E2 0, E3 0, E4 0} C_DIS
LIN {X 805.903, Y 105.862, Z 412, A 0, B 90, C -0, E1 0, E2 0, E3 0, E4 0} C_DIS
LIN {X 807.872, Y 104.951, Z 412, A 0, B 90, C -0, E1 0, E2 0, E3 0, E4 0} C_DIS
LIN {X 809.812, Y 103.978, Z 412, A 0, B 90, C -0, E1 0, E2 0, E3 0, E4 0} C_DIS
LIN {X 811.721, Y 102.945, Z 412, A 0, B 90, C -0, E1 0, E2 0, E3 0, E4 0} C_DIS
LIN {X 813.596, Y 101.852, Z 412, A 0, B 90, C -0, E1 0, E2 0, E3 0, E4 0} C_DIS
LIN {X 815.435, Y 100.701, Z 412, A 0, B 90, C -0, E1 0, E2 0, E3 0, E4 0} C_DIS
LIN {X 817.238, Y 99.493, Z 412, A 0, B 90, C -0, E1 0, E2 0, E3 0, E4 0} C_DIS
LIN {X 819.002, Y 98.229, Z 412, A 0, B 90, C -0, E1 0, E2 0, E3 0, E4 0} C_DIS
LIN {X 820.725, Y 96.91, Z 412, A 0, B 90, C -0, E1 0, E2 0, E3 0, E4 0} C_DIS
LIN {X 822.406, Y 95.537, Z 412, A 0, B 90, C -0, E1 0, E2 0, E3 0, E4 0} C_DIS
LIN {X 824.043, Y 94.112, Z 412, A 0, B 90, C -0, E1 0, E2 0, E3 0, E4 0} C_DIS
LIN {X 825.635, Y 92.637, Z 412, A 0, B 90, C -0, E1 0, E2 0, E3 0, E4 0} C_DIS
LIN {X 827.179, Y 91.112, Z 412, A 0, B 90, C -0, E1 0, E2 0, E3 0, E4 0} C_DIS
LIN {X 828.675, Y 89.54, Z 412, A 0, B 90, C -0, E1 0, E2 0, E3 0, E4 0} C_DIS
LIN {X 830.121, Y 87.921, Z 412, A 0, B 90, C -0, E1 0, E2 0, E3 0, E4 0} C_DIS
LIN {X 831.515, Y 86.258, Z 412, A 0, B 90, C -0, E1 0, E2 0, E3 0, E4 0} C_DIS
LIN {X 832.856, Y 84.552, Z 412, A 0, B 90, C -0, E1 0, E2 0, E3 0, E4 0} C_DIS
LIN {X 834.143, Y 82.805, Z 412, A 0, B 90, C -0, E1 0, E2 0, E3 0, E4 0} C_DIS
LIN {X 835.374, Y 81.018, Z 412, A 0, B 90, C -0, E1 0, E2 0, E3 0, E4 0} C_DIS
LIN {X 836.548, Y 79.193, Z 412, A 0, B 90, C -0, E1 0, E2 0, E3 0, E4 0} C_DIS
LIN {X 837.665, Y 77.332, Z 412, A 0, B 90, C -0, E1 0, E2 0, E3 0, E4 0} C_DIS
LIN {X 838.723, Y 75.437, Z 412, A 0, B 90, C -0, E1 0, E2 0, E3 0, E4 0} C_DIS
LIN {X 839.72, Y 73.51, Z 412, A 0, B 90, C -0, E1 0, E2 0, E3 0, E4 0} C_DIS
LIN {X 840.657, Y 71.552, Z 412, A 0, B 90, C -0, E1 0, E2 0, E3 0, E4 0} C_DIS
LIN {X 841.532, Y 69.566, Z 412, A 0, B 90, C -0, E1 0, E2 0, E3 0, E4 0} C_DIS
LIN {X 842.344, Y 67.553, Z 412, A 0, B 90, C -0, E1 0, E2 0, E3 0, E4 0} C_DIS
LIN {X 843.092, Y 65.516, Z 412, A 0, B 90, C -0, E1 0, E2 0, E3 0, E4 0} C_DIS
LIN {X 843.776, Y 63.457, Z 412, A 0, B 90, C -0, E1 0, E2 0, E3 0, E4 0} C_DIS
LIN {X 844.394, Y 61.377, Z 412, A 0, B 90, C -0, E1 0, E2 0, E3 0, E4 0} C_DIS
LIN {X 844.948, Y 59.278, Z 412, A 0, B 90, C -0, E1 0, E2 0, E3 0, E4 0} C_DIS
LIN {X 845.435, Y 57.163, Z 412, A 0, B 90, C -0, E1 0, E2 0, E3 0, E4 0} C_DIS
LIN {X 845.855, Y 55.034, Z 412, A 0, B 90, C -0, E1 0, E2 0, E3 0, E4 0} C_DIS
LIN {X 846.208, Y 52.893, Z 412, A 0, B 90, C -0, E1 0, E2 0, E3 0, E4 0} C_DIS
LIN {X 846.494, Y 50.742, Z 412, A 0, B 90, C -0, E1 0, E2 0, E3 0, E4 0} C_DIS
LIN {X 846.712, Y 48.583, Z 412, A 0, B 90, C -0, E1 0, E2 0, E3 0, E4 0} C_DIS
LIN {X 846.862, Y 46.418, Z 412, A 0, B 90, C -0, E1 0, E2 0, E3 0, E4 0} C_DIS
LIN {X 846.945, Y 44.249, Z 412, A 0, B 90, C -0, E1 0, E2 0, E3 0, E4 0} C_DIS
LIN {X 846.958, Y 42.079, Z 412, A 0, B 90, C -0, E1 0, E2 0, E3 0, E4 0} C_DIS
LIN {X 846.904, Y 39.909, Z 412, A 0, B 90, C -0, E1 0, E2 0, E3 0, E4 0} C_DIS
LIN {X 846.782, Y 37.743, Z 412, A 0, B 90, C -0, E1 0, E2 0, E3 0, E4 0} C_DIS
LIN {X 846.592, Y 35.581, Z 412, A 0, B 90, C -0, E1 0, E2 0, E3 0, E4 0} C_DIS
LIN {X 846.333, Y 33.426, Z 412, A 0, B 90, C -0, E1 0, E2 0, E3 0, E4 0} C_DIS
LIN {X 846.008, Y 31.28, Z 412, A 0, B 90, C -0, E1 0, E2 0, E3 0, E4 0} C_DIS
LIN {X 845.615, Y 29.146, Z 412, A 0, B 90, C -0, E1 0, E2 0, E3 0, E4 0} C_DIS
LIN {X 845.155, Y 27.025, Z 412, A 0, B 90, C -0, E1 0, E2 0, E3 0, E4 0} C_DIS
LIN {X 844.629, Y 24.92, Z 412, A 0, B 90, C -0, E1 0, E2 0, E3 0, E4 0} C_DIS
LIN {X 844.037, Y 22.832, Z 412, A 0, B 90, C -0, E1 0, E2 0, E3 0, E4 0} C_DIS
LIN {X 843.379, Y 20.764, Z 412, A 0, B 90, C -0, E1 0, E2 0, E3 0, E4 0} C_DIS
LIN {X 842.657, Y 18.717, Z 412, A 0, B 90, C -0, E1 0, E2 0, E3 0, E4 0} C_DIS
LIN {X 841.871, Y 16.694, Z 412, A 0, B 90, C -0, E1 0, E2 0, E3 0, E4 0} C_DIS
LIN {X 841.022, Y 14.697, Z 412, A 0, B 90, C -0, E1 0, E2 0, E3 0, E4 0} C_DIS
LIN {X 840.111, Y 12.728, Z 412, A 0, B 90, C -0, E1 0, E2 0, E3 0, E4 0} C_DIS
LIN {X 839.138, Y 10.788, Z 412, A 0, B 90, C -0, E1 0, E2 0, E3 0, E4 0} C_DIS
LIN {X 838.105, Y 8.879, Z 412, A 0, B 90, C -0, E1 0, E2 0, E3 0, E4 0} C_DIS
LIN {X 837.012, Y 7.004, Z 412, A 0, B 90, C -0, E1 0, E2 0, E3 0, E4 0} C_DIS
LIN {X 835.861, Y 5.165, Z 412, A 0, B 90, C -0, E1 0, E2 0, E3 0, E4 0} C_DIS
LIN {X 834.653, Y 3.362, Z 412, A 0, B 90, C -0, E1 0, E2 0, E3 0, E4 0} C_DIS
LIN {X 833.389, Y 1.598, Z 412, A 0, B 90, C -0, E1 0, E2 0, E3 0, E4 0} C_DIS
LIN {X 832.07, Y -0.125, Z 412, A 0, B 90, C -0, E1 0, E2 0, E3 0, E4 0} C_DIS
LIN {X 830.697, Y -1.806, Z 412, A 0, B 90, C -0, E1 0, E2 0, E3 0, E4 0} C_DIS
LIN {X 829.272, Y -3.443, Z 412, A 0, B 90, C -0, E1 0, E2 0, E3 0, E4 0} C_DIS
LIN {X 827.797, Y -5.035, Z 412, A 0, B 90, C -0, E1 0, E2 0, E3 0, E4 0} C_DIS
LIN {X 826.272, Y -6.579, Z 412, A 0, B 90, C -0, E1 0, E2 0, E3 0, E4 0} C_DIS
LIN {X 824.7, Y -8.075, Z 412, A 0, B 90, C -0, E1 0, E2 0, E3 0, E4 0} C_DIS
LIN {X 823.081, Y -9.521, Z 412, A 0, B 90, C -0, E1 0, E2 0, E3 0, E4 0} C_DIS
LIN {X 821.418, Y -10.915, Z 412, A 0, B 90, C -0, E1 0, E2 0, E3 0, E4 0} C_DIS
LIN {X 819.712, Y -12.256, Z 412, A 0, B 90, C -0, E1 0, E2 0, E3 0, E4 0} C_DIS
LIN {X 817.965, Y -13.543, Z 412, A 0, B 90, C -0, E1 0, E2 0, E3 0, E4 0} C_DIS
LIN {X 816.178, Y -14.774, Z 412, A 0, B 90, C -0, E1 0, E2 0, E3 0, E4 0} C_DIS
LIN {X 814.353, Y -15.948, Z 412, A 0, B 90, C -0, E1 0, E2 0, E3 0, E4 0} C_DIS
LIN {X 812.492, Y -17.065, Z 412, A 0, B 90, C -0, E1 0, E2 0, E3 0, E4 0} C_DIS
LIN {X 810.597, Y -18.123, Z 412, A 0, B 90, C -0, E1 0, E2 0, E3 0, E4 0} C_DIS
LIN {X 808.67, Y -19.12, Z 412, A 0, B 90, C -0, E1 0, E2 0, E3 0, E4 0} C_DIS
LIN {X 806.712, Y -20.057, Z 412, A 0, B 90, C -0, E1 0, E2 0, E3 0, E4 0} C_DIS
LIN {X 804.726, Y -20.932, Z 412, A 0, B 90, C -0, E1 0, E2 0, E3 0, E4 0} C_DIS
LIN {X 802.713, Y -21.744, Z 412, A 0, B 90, C -0, E1 0, E2 0, E3 0, E4 0} C_DIS
LIN {X 800.676, Y -22.492, Z 412, A 0, B 90, C -0, E1 0, E2 0, E3 0, E4 0} C_DIS
LIN {X 798.617, Y -23.176, Z 412, A 0, B 90, C -0, E1 0, E2 0, E3 0, E4 0} C_DIS
LIN {X 796.537, Y -23.794, Z 412, A 0, B 90, C -0, E1 0, E2 0, E3 0, E4 0} C_DIS
LIN {X 794.438, Y -24.348, Z 412, A 0, B 90, C -0, E1 0, E2 0, E3 0, E4 0} C_DIS
LIN {X 792.323, Y -24.835, Z 412, A 0, B 90, C -0, E1 0, E2 0, E3 0, E4 0} C_DIS
LIN {X 790.194, Y -25.255, Z 412, A 0, B 90, C -0, E1 0, E2 0, E3 0, E4 0} C_DIS
LIN {X 788.053, Y -25.608, Z 412, A 0, B 90, C -0, E1 0, E2 0, E3 0, E4 0} C_DIS
LIN {X 785.902, Y -25.894, Z 412, A 0, B 90, C -0, E1 0, E2 0, E3 0, E4 0} C_DIS
LIN {X 783.742, Y -26.112, Z 412, A 0, B 90, C -0, E1 0, E2 0, E3 0, E4 0} C_DIS
LIN {X 781.578, Y -26.262, Z 412, A 0, B 90, C -0, E1 0, E2 0, E3 0, E4 0} C_DIS
LIN {X 779.409, Y -26.344, Z 412, A 0, B 90, C -0, E1 0, E2 0, E3 0, E4 0} C_DIS
LIN {X 777.239, Y -26.358, Z 412, A 0, B 90, C -0, E1 0, E2 0, E3 0, E4 0} C_DIS
LIN {X 775.069, Y -26.304, Z 412, A 0, B 90, C -0, E1 0, E2 0, E3 0, E4 0} C_DIS
LIN {X 772.903, Y -26.182, Z 412, A 0, B 90, C -0, E1 0, E2 0, E3 0, E4 0} C_DIS
LIN {X 770.741, Y -25.992, Z 412, A 0, B 90, C -0, E1 0, E2 0, E3 0, E4 0} C_DIS
LIN {X 768.586, Y -25.733, Z 412, A 0, B 90, C -0, E1 0, E2 0, E3 0, E4 0} C_DIS
LIN {X 766.44, Y -25.408, Z 412, A 0, B 90, C -0, E1 0, E2 0, E3 0, E4 0} C_DIS
LIN {X 764.306, Y -25.015, Z 412, A 0, B 90, C -0, E1 0, E2 0, E3 0, E4 0} C_DIS
LIN {X 762.185, Y -24.555, Z 412, A 0, B 90, C -0, E1 0, E2 0, E3 0, E4 0} C_DIS
LIN {X 760.08, Y -24.029, Z 412, A 0, B 90, C -0, E1 0, E2 0, E3 0, E4 0} C_DIS
LIN {X 757.992, Y -23.437, Z 412, A 0, B 90, C -0, E1 0, E2 0, E3 0, E4 0} C_DIS
LIN {X 755.924, Y -22.779, Z 412, A 0, B 90, C -0, E1 0, E2 0, E3 0, E4 0} C_DIS
LIN {X 753.877, Y -22.057, Z 412, A 0, B 90, C -0, E1 0, E2 0, E3 0, E4 0} C_DIS
LIN {X 751.854, Y -21.271, Z 412, A 0, B 90, C -0, E1 0, E2 0, E3 0, E4 0} C_DIS
LIN {X 749.857, Y -20.422, Z 412, A 0, B 90, C -0, E1 0, E2 0, E3 0, E4 0} C_DIS
LIN {X 747.888, Y -19.511, Z 412, A 0, B 90, C -0, E1 0, E2 0, E3 0, E4 0} C_DIS
LIN {X 745.948, Y -18.538, Z 412, A 0, B 90, C -0, E1 0, E2 0, E3 0, E4 0} C_DIS
LIN {X 744.039, Y -17.505, Z 412, A 0, B 90, C -0, E1 0, E2 0, E3 0, E4 0} C_DIS
LIN {X 742.164, Y -16.412, Z 412, A 0, B 90, C -0, E1 0, E2 0, E3 0, E4 0} C_DIS
LIN {X 740.325, Y -15.261, Z 412, A 0, B 90, C -0, E1 0, E2 0, E3 0, E4 0} C_DIS
LIN {X 738.522, Y -14.053, Z 412, A 0, B 90, C -0, E1 0, E2 0, E3 0, E4 0} C_DIS
LIN {X 736.758, Y -12.789, Z 412, A 0, B 90, C -0, E1 0, E2 0, E3 0, E4 0} C_DIS
LIN {X 735.035, Y -11.47, Z 412, A 0, B 90, C -0, E1 0, E2 0, E3 0, E4 0} C_DIS
LIN {X 733.354, Y -10.097, Z 412, A 0, B 90, C -0, E1 0, E2 0, E3 0, E4 0} C_DIS
LIN {X 731.717, Y -8.672, Z 412, A 0, B 90, C -0, E1 0, E2 0, E3 0, E4 0} C_DIS
LIN {X 730.125, Y -7.197, Z 412, A 0, B 90, C -0, E1 0, E2 0, E3 0, E4 0} C_DIS
LIN {X 728.581, Y -5.672, Z 412, A 0, B 90, C -0, E1 0, E2 0, E3 0, E4 0} C_DIS
LIN {X 727.085, Y -4.1, Z 412, A 0, B 90, C -0, E1 0, E2 0, E3 0, E4 0} C_DIS
LIN {X 725.639, Y -2.481, Z 412, A 0, B 90, C -0, E1 0, E2 0, E3 0, E4 0} C_DIS
LIN {X 724.245, Y -0.818, Z 412, A 0, B 90, C -0, E1 0, E2 0, E3 0, E4 0} C_DIS
LIN {X 722.904, Y 0.888, Z 412, A 0, B 90, C -0, E1 0, E2 0, E3 0, E4 0} C_DIS
LIN {X 721.617, Y 2.635, Z 412, A 0, B 90, C -0, E1 0, E2 0, E3 0, E4 0} C_DIS
LIN {X 720.386, Y 4.422, Z 412, A 0, B 90, C -0, E1 0, E2 0, E3 0, E4 0} C_DIS
LIN {X 719.212, Y 6.247, Z 412, A 0, B 90, C -0, E1 0, E2 0, E3 0, E4 0} C_DIS
LIN {X 718.095, Y 8.108, Z 412, A 0, B 90, C -0, E1 0, E2 0, E3 0, E4 0} C_DIS
LIN {X 717.037, Y 10.003, Z 412, A 0, B 90, C -0, E1 0, E2 0, E3 0, E4 0} C_DIS
LIN {X 716.04, Y 11.93, Z 412, A 0, B 90, C -0, E1 0, E2 0, E3 0, E4 0} C_DIS
LIN {X 715.103, Y 13.888, Z 412, A 0, B 90, C -0, E1 0, E2 0, E3 0, E4 0} C_DIS
LIN {X 714.228, Y 15.874, Z 412, A 0, B 90, C -0, E1 0, E2 0, E3 0, E4 0} C_DIS
LIN {X 713.416, Y 17.887, Z 412, A 0, B 90, C -0, E1 0, E2 0, E3 0, E4 0} C_DIS
LIN {X 712.668, Y 19.924, Z 412, A 0, B 90, C -0, E1 0, E2 0, E3 0, E4 0} C_DIS
LIN {X 711.984, Y 21.983, Z 412, A 0, B 90, C -0, E1 0, E2 0, E3 0, E4 0} C_DIS
LIN {X 711.366, Y 24.063, Z 412, A 0, B 90, C -0, E1 0, E2 0, E3 0, E4 0} C_DIS
LIN {X 710.812, Y 26.162, Z 412, A 0, B 90, C -0, E1 0, E2 0, E3 0, E4 0} C_DIS
LIN {X 710.325, Y 28.277, Z 412, A 0, B 90, C -0, E1 0, E2 0, E3 0, E4 0} C_DIS
LIN {X 709.905, Y 30.406, Z 412, A 0, B 90, C -0, E1 0, E2 0, E3 0, E4 0} C_DIS
LIN {X 709.552, Y 32.547, Z 412, A 0, B 90, C -0, E1 0, E2 0, E3 0, E4 0} C_DIS
LIN {X 709.266, Y 34.698, Z 412, A 0, B 90, C -0, E1 0, E2 0, E3 0, E4 0} C_DIS
LIN {X 709.048, Y 36.857, Z 412, A 0, B 90, C -0, E1 0, E2 0, E3 0, E4 0} C_DIS
LIN {X 708.898, Y 39.022, Z 412, A 0, B 90, C -0, E1 0, E2 0, E3 0, E4 0} C_DIS
LIN {X 708.815, Y 41.191, Z 412, A 0, B 90, C -0, E1 0, E2 0, E3 0, E4 0} C_DIS
LIN {X 708.802, Y 43.361, Z 412, A 0, B 90, C -0, E1 0, E2 0, E3 0, E4 0} C_DIS
LIN {X 708.856, Y 45.531, Z 412, A 0, B 90, C -0, E1 0, E2 0, E3 0, E4 0} C_DIS
LIN {X 708.978, Y 47.697, Z 412, A 0, B 90, C -0, E1 0, E2 0, E3 0, E4 0} C_DIS
LIN {X 709.168, Y 49.859, Z 412, A 0, B 90, C -0, E1 0, E2 0, E3 0, E4 0} C_DIS
LIN {X 709.427, Y 52.014, Z 412, A 0, B 90, C -0, E1 0, E2 0, E3 0, E4 0} C_DIS
LIN {X 709.752, Y 54.16, Z 412, A 0, B 90, C -0, E1 0, E2 0, E3 0, E4 0} C_DIS
LIN {X 710.145, Y 56.294, Z 412, A 0, B 90, C -0, E1 0, E2 0, E3 0, E4 0} C_DIS
LIN {X 710.605, Y 58.415, Z 412, A 0, B 90, C -0, E1 0, E2 0, E3 0, E4 0} C_DIS
LIN {X 711.131, Y 60.52, Z 412, A 0, B 90, C -0, E1 0, E2 0, E3 0, E4 0} C_DIS
LIN {X 711.723, Y 62.608, Z 412, A 0, B 90, C -0, E1 0, E2 0, E3 0, E4 0} C_DIS
LIN {X 712.571, Y 64.058, Z 414, A 0, B 90, C -0, E1 0, E2 0, E3 0, E4 0} C_DIS
LIN {X 713.274, Y 66.099, Z 414, A 0, B 90, C -0, E1 0, E2 0, E3 0, E4 0} C_DIS
LIN {X 714.04, Y 68.116, Z 414, A 0, B 90, C -0, E1 0, E2 0, E3 0, E4 0} C_DIS
LIN {X 714.869, Y 70.109, Z 414, A 0, B 90, C -0, E1 0, E2 0, E3 0, E4 0} C_DIS
LIN {X 715.76, Y 72.075, Z 414, A 0, B 90, C -0, E1 0, E2 0, E3 0, E4 0} C_DIS
LIN {X 716.713, Y 74.012, Z 414, A 0, B 90, C -0, E1 0, E2 0, E3 0, E4 0} C_DIS
LIN {X 717.726, Y 75.917, Z 414, A 0, B 90, C -0, E1 0, E2 0, E3 0, E4 0} C_DIS
LIN {X 718.799, Y 77.791, Z 414, A 0, B 90, C -0, E1 0, E2 0, E3 0, E4 0} C_DIS
LIN {X 719.929, Y 79.629, Z 414, A 0, B 90, C -0, E1 0, E2 0, E3 0, E4 0} C_DIS
LIN {X 721.117, Y 81.431, Z 414, A 0, B 90, C -0, E1 0, E2 0, E3 0, E4 0} C_DIS
LIN {X 722.361, Y 83.195, Z 414, A 0, B 90, C -0, E1 0, E2 0, E3 0, E4 0} C_DIS
LIN {X 723.66, Y 84.919, Z 414, A 0, B 90, C -0, E1 0, E2 0, E3 0, E4 0} C_DIS
LIN {X 725.012, Y 86.601, Z 414, A 0, B 90, C -0, E1 0, E2 0, E3 0, E4 0} C_DIS
LIN {X 726.417, Y 88.24, Z 414, A 0, B 90, C -0, E1 0, E2 0, E3 0, E4 0} C_DIS
LIN {X 727.872, Y 89.834, Z 414, A 0, B 90, C -0, E1 0, E2 0, E3 0, E4 0} C_DIS
LIN {X 729.376, Y 91.382, Z 414, A 0, B 90, C -0, E1 0, E2 0, E3 0, E4 0} C_DIS
LIN {X 730.929, Y 92.881, Z 414, A 0, B 90, C -0, E1 0, E2 0, E3 0, E4 0} C_DIS
LIN {X 732.528, Y 94.331, Z 414, A 0, B 90, C -0, E1 0, E2 0, E3 0, E4 0} C_DIS
LIN {X 734.171, Y 95.73, Z 414, A 0, B 90, C -0, E1 0, E2 0, E3 0, E4 0} C_DIS
LIN {X 735.858, Y 97.077, Z 414, A 0, B 90, C -0, E1 0, E2 0, E3 0, E4 0} C_DIS
LIN {X 737.586, Y 98.37, Z 414, A 0, B 90, C -0, E1 0, E2 0, E3 0, E4 0} C_DIS
LIN {X 739.354, Y 99.608, Z 414, A 0, B 90, C -0, E1 0, E2 0, E3 0, E4 0} C_DIS
LIN {X 741.16, Y 100.79, Z 414, A 0, B 90, C -0, E1 0, E2 0, E3 0, E4 0} C_DIS
LIN {X 743.002, Y 101.915, Z 414, A 0, B 90, C -0, E1 0, E2 0, E3 0, E4 0} C_DIS
LIN {X 744.879, Y 102.982, Z 414, A 0, B 90, C -0, E1 0, E2 0, E3 0, E4 0} C_DIS
LIN {X 746.788, Y 103.988, Z 414, A 0, B 90, C -0, E1 0, E2 0, E3 0, E4 0} C_DIS
LIN {X 748.728, Y 104.935, Z 414, A 0, B 90, C -0, E1 0, E2 0, E3 0, E4 0} C_DIS
LIN {X 750.696, Y 105.82, Z 414, A 0, B 90, C -0, E1 0, E2 0, E3 0, E4 0} C_DIS
LIN {X 752.692, Y 106.643, Z 414, A 0, B 90, C -0, E1 0, E2 0, E3 0, E4 0} C_DIS
LIN {X 754.712, Y 107.402, Z 414, A 0, B 90, C -0, E1 0, E2 0, E3 0, E4 0} C_DIS
LIN {X 756.755, Y 108.098, Z 414, A 0, B 90, C -0, E1 0, E2 0, E3 0, E4 0} C_DIS
LIN {X 758.819, Y 108.729, Z 414, A 0, B 90, C -0, E1 0, E2 0, E3 0, E4 0} C_DIS
LIN {X 760.902, Y 109.295, Z 414, A 0, B 90, C -0, E1 0, E2 0, E3 0, E4 0} C_DIS
LIN {X 763.001, Y 109.796, Z 414, A 0, B 90, C -0, E1 0, E2 0, E3 0, E4 0} C_DIS
LIN {X 765.116, Y 110.23, Z 414, A 0, B 90, C -0, E1 0, E2 0, E3 0, E4 0} C_DIS
LIN {X 767.242, Y 110.598, Z 414, A 0, B 90, C -0, E1 0, E2 0, E3 0, E4 0} C_DIS
LIN {X 769.38, Y 110.898, Z 414, A 0, B 90, C -0, E1 0, E2 0, E3 0, E4 0} C_DIS
LIN {X 771.526, Y 111.132, Z 414, A 0, B 90, C -0, E1 0, E2 0, E3 0, E4 0} C_DIS
LIN {X 773.677, Y 111.298, Z 414, A 0, B 90, C -0, E1 0, E2 0, E3 0, E4 0} C_DIS
LIN {X 775.834, Y 111.396, Z 414, A 0, B 90, C -0, E1 0, E2 0, E3 0, E4 0} C_DIS
LIN {X 777.992, Y 111.426, Z 414, A 0, B 90, C -0, E1 0, E2 0, E3 0, E4 0} C_DIS
LIN {X 780.15, Y 111.389, Z 414, A 0, B 90, C -0, E1 0, E2 0, E3 0, E4 0} C_DIS
LIN {X 782.306, Y 111.284, Z 414, A 0, B 90, C -0, E1 0, E2 0, E3 0, E4 0} C_DIS
LIN {X 784.457, Y 111.111, Z 414, A 0, B 90, C -0, E1 0, E2 0, E3 0, E4 0} C_DIS
LIN {X 786.602, Y 110.87, Z 414, A 0, B 90, C -0, E1 0, E2 0, E3 0, E4 0} C_DIS
LIN {X 788.738, Y 110.563, Z 414, A 0, B 90, C -0, E1 0, E2 0, E3 0, E4 0} C_DIS
LIN {X 790.864, Y 110.188, Z 414, A 0, B 90, C -0, E1 0, E2 0, E3 0, E4 0} C_DIS
LIN {X 792.977, Y 109.747, Z 414, A 0, B 90, C -0, E1 0, E2 0, E3 0, E4 0} C_DIS
LIN {X 795.075, Y 109.24, Z 414, A 0, B 90, C -0, E1 0, E2 0, E3 0, E4 0} C_DIS
LIN {X 797.156, Y 108.667, Z 414, A 0, B 90, C -0, E1 0, E2 0, E3 0, E4 0} C_DIS
LIN {X 799.218, Y 108.029, Z 414, A 0, B 90, C -0, E1 0, E2 0, E3 0, E4 0} C_DIS
LIN {X 801.259, Y 107.326, Z 414, A 0, B 90, C -0, E1 0, E2 0, E3 0, E4 0} C_DIS
LIN {X 803.276, Y 106.56, Z 414, A 0, B 90, C -0, E1 0, E2 0, E3 0, E4 0} C_DIS
LIN {X 805.269, Y 105.731, Z 414, A 0, B 90, C -0, E1 0, E2 0, E3 0, E4 0} C_DIS
LIN {X 807.235, Y 104.84, Z 414, A 0, B 90, C -0, E1 0, E2 0, E3 0, E4 0} C_DIS
LIN {X 809.172, Y 103.887, Z 414, A 0, B 90, C -0, E1 0, E2 0, E3 0, E4 0} C_DIS
LIN {X 811.077, Y 102.874, Z 414, A 0, B 90, C -0, E1 0, E2 0, E3 0, E4 0} C_DIS
LIN {X 812.951, Y 101.801, Z 414, A 0, B 90, C -0, E1 0, E2 0, E3 0, E4 0} C_DIS
LIN {X 814.789, Y 100.671, Z 414, A 0, B 90, C -0, E1 0, E2 0, E3 0, E4 0} C_DIS
LIN {X 816.591, Y 99.483, Z 414, A 0, B 90, C -0, E1 0, E2 0, E3 0, E4 0} C_DIS
LIN {X 818.355, Y 98.239, Z 414, A 0, B 90, C -0, E1 0, E2 0, E3 0, E4 0} C_DIS
LIN {X 820.079, Y 96.94, Z 414, A 0, B 90, C -0, E1 0, E2 0, E3 0, E4 0} C_DIS
LIN {X 821.761, Y 95.588, Z 414, A 0, B 90, C -0, E1 0, E2 0, E3 0, E4 0} C_DIS
LIN {X 823.4, Y 94.183, Z 414, A 0, B 90, C -0, E1 0, E2 0, E3 0, E4 0} C_DIS
LIN {X 824.994, Y 92.728, Z 414, A 0, B 90, C -0, E1 0, E2 0, E3 0, E4 0} C_DIS
LIN {X 826.542, Y 91.224, Z 414, A 0, B 90, C -0, E1 0, E2 0, E3 0, E4 0} C_DIS
LIN {X 828.041, Y 89.671, Z 414, A 0, B 90, C -0, E1 0, E2 0, E3 0, E4 0} C_DIS
LIN {X 829.491, Y 88.072, Z 414, A 0, B 90, C -0, E1 0, E2 0, E3 0, E4 0} C_DIS
LIN {X 830.89, Y 86.429, Z 414, A 0, B 90, C -0, E1 0, E2 0, E3 0, E4 0} C_DIS
LIN {X 832.237, Y 84.742, Z 414, A 0, B 90, C -0, E1 0, E2 0, E3 0, E4 0} C_DIS
LIN {X 833.53, Y 83.014, Z 414, A 0, B 90, C -0, E1 0, E2 0, E3 0, E4 0} C_DIS
LIN {X 834.768, Y 81.246, Z 414, A 0, B 90, C -0, E1 0, E2 0, E3 0, E4 0} C_DIS
LIN {X 835.95, Y 79.44, Z 414, A 0, B 90, C -0, E1 0, E2 0, E3 0, E4 0} C_DIS
LIN {X 837.075, Y 77.598, Z 414, A 0, B 90, C -0, E1 0, E2 0, E3 0, E4 0} C_DIS
LIN {X 838.142, Y 75.721, Z 414, A 0, B 90, C -0, E1 0, E2 0, E3 0, E4 0} C_DIS
LIN {X 839.148, Y 73.812, Z 414, A 0, B 90, C -0, E1 0, E2 0, E3 0, E4 0} C_DIS
LIN {X 840.095, Y 71.872, Z 414, A 0, B 90, C -0, E1 0, E2 0, E3 0, E4 0} C_DIS
LIN {X 840.98, Y 69.904, Z 414, A 0, B 90, C -0, E1 0, E2 0, E3 0, E4 0} C_DIS
LIN {X 841.803, Y 67.908, Z 414, A 0, B 90, C -0, E1 0, E2 0, E3 0, E4 0} C_DIS
LIN {X 842.562, Y 65.888, Z 414, A 0, B 90, C -0, E1 0, E2 0, E3 0, E4 0} C_DIS
LIN {X 843.258, Y 63.845, Z 414, A 0, B 90, C -0, E1 0, E2 0, E3 0, E4 0} C_DIS
LIN {X 843.889, Y 61.781, Z 414, A 0, B 90, C -0, E1 0, E2 0, E3 0, E4 0} C_DIS
LIN {X 844.455, Y 59.698, Z 414, A 0, B 90, C -0, E1 0, E2 0, E3 0, E4 0} C_DIS
LIN {X 844.956, Y 57.599, Z 414, A 0, B 90, C -0, E1 0, E2 0, E3 0, E4 0} C_DIS
LIN {X 845.39, Y 55.484, Z 414, A 0, B 90, C -0, E1 0, E2 0, E3 0, E4 0} C_DIS
LIN {X 845.758, Y 53.358, Z 414, A 0, B 90, C -0, E1 0, E2 0, E3 0, E4 0} C_DIS
LIN {X 846.058, Y 51.22, Z 414, A 0, B 90, C -0, E1 0, E2 0, E3 0, E4 0} C_DIS
LIN {X 846.292, Y 49.074, Z 414, A 0, B 90, C -0, E1 0, E2 0, E3 0, E4 0} C_DIS
LIN {X 846.458, Y 46.922, Z 414, A 0, B 90, C -0, E1 0, E2 0, E3 0, E4 0} C_DIS
LIN {X 846.556, Y 44.766, Z 414, A 0, B 90, C -0, E1 0, E2 0, E3 0, E4 0} C_DIS
LIN {X 846.586, Y 42.608, Z 414, A 0, B 90, C -0, E1 0, E2 0, E3 0, E4 0} C_DIS
LIN {X 846.549, Y 40.45, Z 414, A 0, B 90, C -0, E1 0, E2 0, E3 0, E4 0} C_DIS
LIN {X 846.444, Y 38.294, Z 414, A 0, B 90, C -0, E1 0, E2 0, E3 0, E4 0} C_DIS
LIN {X 846.271, Y 36.143, Z 414, A 0, B 90, C -0, E1 0, E2 0, E3 0, E4 0} C_DIS
LIN {X 846.03, Y 33.998, Z 414, A 0, B 90, C -0, E1 0, E2 0, E3 0, E4 0} C_DIS
LIN {X 845.723, Y 31.862, Z 414, A 0, B 90, C -0, E1 0, E2 0, E3 0, E4 0} C_DIS
LIN {X 845.348, Y 29.736, Z 414, A 0, B 90, C -0, E1 0, E2 0, E3 0, E4 0} C_DIS
LIN {X 844.907, Y 27.623, Z 414, A 0, B 90, C -0, E1 0, E2 0, E3 0, E4 0} C_DIS
LIN {X 844.4, Y 25.525, Z 414, A 0, B 90, C -0, E1 0, E2 0, E3 0, E4 0} C_DIS
LIN {X 843.827, Y 23.444, Z 414, A 0, B 90, C -0, E1 0, E2 0, E3 0, E4 0} C_DIS
LIN {X 843.189, Y 21.382, Z 414, A 0, B 90, C -0, E1 0, E2 0, E3 0, E4 0} C_DIS
LIN {X 842.486, Y 19.341, Z 414, A 0, B 90, C -0, E1 0, E2 0, E3 0, E4 0} C_DIS
LIN {X 841.72, Y 17.324, Z 414, A 0, B 90, C -0, E1 0, E2 0, E3 0, E4 0} C_DIS
LIN {X 840.891, Y 15.331, Z 414, A 0, B 90, C -0, E1 0, E2 0, E3 0, E4 0} C_DIS
LIN {X 840, Y 13.365, Z 414, A 0, B 90, C -0, E1 0, E2 0, E3 0, E4 0} C_DIS
LIN {X 839.047, Y 11.428, Z 414, A 0, B 90, C -0, E1 0, E2 0, E3 0, E4 0} C_DIS
LIN {X 838.034, Y 9.523, Z 414, A 0, B 90, C -0, E1 0, E2 0, E3 0, E4 0} C_DIS
LIN {X 836.961, Y 7.649, Z 414, A 0, B 90, C -0, E1 0, E2 0, E3 0, E4 0} C_DIS
LIN {X 835.831, Y 5.811, Z 414, A 0, B 90, C -0, E1 0, E2 0, E3 0, E4 0} C_DIS
LIN {X 834.643, Y 4.009, Z 414, A 0, B 90, C -0, E1 0, E2 0, E3 0, E4 0} C_DIS
LIN {X 833.399, Y 2.245, Z 414, A 0, B 90, C -0, E1 0, E2 0, E3 0, E4 0} C_DIS
LIN {X 832.1, Y 0.521, Z 414, A 0, B 90, C -0, E1 0, E2 0, E3 0, E4 0} C_DIS
LIN {X 830.748, Y -1.161, Z 414, A 0, B 90, C -0, E1 0, E2 0, E3 0, E4 0} C_DIS
LIN {X 829.343, Y -2.8, Z 414, A 0, B 90, C -0, E1 0, E2 0, E3 0, E4 0} C_DIS
LIN {X 827.888, Y -4.394, Z 414, A 0, B 90, C -0, E1 0, E2 0, E3 0, E4 0} C_DIS
LIN {X 826.383, Y -5.942, Z 414, A 0, B 90, C -0, E1 0, E2 0, E3 0, E4 0} C_DIS
LIN {X 824.831, Y -7.441, Z 414, A 0, B 90, C -0, E1 0, E2 0, E3 0, E4 0} C_DIS
LIN {X 823.232, Y -8.891, Z 414, A 0, B 90, C -0, E1 0, E2 0, E3 0, E4 0} C_DIS
LIN {X 821.589, Y -10.29, Z 414, A 0, B 90, C -0, E1 0, E2 0, E3 0, E4 0} C_DIS
LIN {X 819.902, Y -11.637, Z 414, A 0, B 90, C -0, E1 0, E2 0, E3 0, E4 0} C_DIS
LIN {X 818.174, Y -12.93, Z 414, A 0, B 90, C -0, E1 0, E2 0, E3 0, E4 0} C_DIS
LIN {X 816.406, Y -14.168, Z 414, A 0, B 90, C -0, E1 0, E2 0, E3 0, E4 0} C_DIS
LIN {X 814.6, Y -15.35, Z 414, A 0, B 90, C -0, E1 0, E2 0, E3 0, E4 0} C_DIS
LIN {X 812.758, Y -16.475, Z 414, A 0, B 90, C -0, E1 0, E2 0, E3 0, E4 0} C_DIS
LIN {X 810.881, Y -17.542, Z 414, A 0, B 90, C -0, E1 0, E2 0, E3 0, E4 0} C_DIS
LIN {X 808.972, Y -18.548, Z 414, A 0, B 90, C -0, E1 0, E2 0, E3 0, E4 0} C_DIS
LIN {X 807.032, Y -19.495, Z 414, A 0, B 90, C -0, E1 0, E2 0, E3 0, E4 0} C_DIS
LIN {X 805.064, Y -20.38, Z 414, A 0, B 90, C -0, E1 0, E2 0, E3 0, E4 0} C_DIS
LIN {X 803.068, Y -21.203, Z 414, A 0, B 90, C -0, E1 0, E2 0, E3 0, E4 0} C_DIS
LIN {X 801.048, Y -21.962, Z 414, A 0, B 90, C -0, E1 0, E2 0, E3 0, E4 0} C_DIS
LIN {X 799.005, Y -22.658, Z 414, A 0, B 90, C -0, E1 0, E2 0, E3 0, E4 0} C_DIS
LIN {X 796.941, Y -23.289, Z 414, A 0, B 90, C -0, E1 0, E2 0, E3 0, E4 0} C_DIS
LIN {X 794.858, Y -23.855, Z 414, A 0, B 90, C -0, E1 0, E2 0, E3 0, E4 0} C_DIS
LIN {X 792.759, Y -24.356, Z 414, A 0, B 90, C -0, E1 0, E2 0, E3 0, E4 0} C_DIS
LIN {X 790.644, Y -24.79, Z 414, A 0, B 90, C -0, E1 0, E2 0, E3 0, E4 0} C_DIS
LIN {X 788.518, Y -25.158, Z 414, A 0, B 90, C -0, E1 0, E2 0, E3 0, E4 0} C_DIS
LIN {X 786.38, Y -25.458, Z 414, A 0, B 90, C -0, E1 0, E2 0, E3 0, E4 0} C_DIS
LIN {X 784.234, Y -25.692, Z 414, A 0, B 90, C -0, E1 0, E2 0, E3 0, E4 0} C_DIS
LIN {X 782.082, Y -25.858, Z 414, A 0, B 90, C -0, E1 0, E2 0, E3 0, E4 0} C_DIS
LIN {X 779.926, Y -25.956, Z 414, A 0, B 90, C -0, E1 0, E2 0, E3 0, E4 0} C_DIS
LIN {X 777.768, Y -25.986, Z 414, A 0, B 90, C -0, E1 0, E2 0, E3 0, E4 0} C_DIS
LIN {X 775.61, Y -25.949, Z 414, A 0, B 90, C -0, E1 0, E2 0, E3 0, E4 0} C_DIS
LIN {X 773.454, Y -25.844, Z 414, A 0, B 90, C -0, E1 0, E2 0, E3 0, E4 0} C_DIS
LIN {X 771.303, Y -25.671, Z 414, A 0, B 90, C -0, E1 0, E2 0, E3 0, E4 0} C_DIS
LIN {X 769.158, Y -25.43, Z 414, A 0, B 90, C -0, E1 0, E2 0, E3 0, E4 0} C_DIS
LIN {X 767.022, Y -25.123, Z 414, A 0, B 90, C -0, E1 0, E2 0, E3 0, E4 0} C_DIS
LIN {X 764.896, Y -24.748, Z 414, A 0, B 90, C -0, E1 0, E2 0, E3 0, E4 0} C_DIS
LIN {X 762.783, Y -24.307, Z 414, A 0, B 90, C -0, E1 0, E2 0, E3 0, E4 0} C_DIS
LIN {X 760.685, Y -23.8, Z 414, A 0, B 90, C -0, E1 0, E2 0, E3 0, E4 0} C_DIS
LIN {X 758.604, Y -23.227, Z 414, A 0, B 90, C -0, E1 0, E2 0, E3 0, E4 0} C_DIS
LIN {X 756.542, Y -22.589, Z 414, A 0, B 90, C -0, E1 0, E2 0, E3 0, E4 0} C_DIS
LIN {X 754.501, Y -21.886, Z 414, A 0, B 90, C -0, E1 0, E2 0, E3 0, E4 0} C_DIS
LIN {X 752.484, Y -21.12, Z 414, A 0, B 90, C -0, E1 0, E2 0, E3 0, E4 0} C_DIS
LIN {X 750.491, Y -20.291, Z 414, A 0, B 90, C -0, E1 0, E2 0, E3 0, E4 0} C_DIS
LIN {X 748.525, Y -19.4, Z 414, A 0, B 90, C -0, E1 0, E2 0, E3 0, E4 0} C_DIS
LIN {X 746.588, Y -18.447, Z 414, A 0, B 90, C -0, E1 0, E2 0, E3 0, E4 0} C_DIS
LIN {X 744.683, Y -17.434, Z 414, A 0, B 90, C -0, E1 0, E2 0, E3 0, E4 0} C_DIS
LIN {X 742.809, Y -16.361, Z 414, A 0, B 90, C -0, E1 0, E2 0, E3 0, E4 0} C_DIS
LIN {X 740.971, Y -15.231, Z 414, A 0, B 90, C -0, E1 0, E2 0, E3 0, E4 0} C_DIS
LIN {X 739.169, Y -14.043, Z 414, A 0, B 90, C -0, E1 0, E2 0, E3 0, E4 0} C_DIS
LIN {X 737.405, Y -12.799, Z 414, A 0, B 90, C -0, E1 0, E2 0, E3 0, E4 0} C_DIS
LIN {X 735.681, Y -11.5, Z 414, A 0, B 90, C -0, E1 0, E2 0, E3 0, E4 0} C_DIS
LIN {X 733.999, Y -10.148, Z 414, A 0, B 90, C -0, E1 0, E2 0, E3 0, E4 0} C_DIS
LIN {X 732.36, Y -8.743, Z 414, A 0, B 90, C -0, E1 0, E2 0, E3 0, E4 0} C_DIS
LIN {X 730.766, Y -7.288, Z 414, A 0, B 90, C -0, E1 0, E2 0, E3 0, E4 0} C_DIS
LIN {X 729.218, Y -5.784, Z 414, A 0, B 90, C -0, E1 0, E2 0, E3 0, E4 0} C_DIS
LIN {X 727.719, Y -4.231, Z 414, A 0, B 90, C -0, E1 0, E2 0, E3 0, E4 0} C_DIS
LIN {X 726.269, Y -2.632, Z 414, A 0, B 90, C -0, E1 0, E2 0, E3 0, E4 0} C_DIS
LIN {X 724.87, Y -0.989, Z 414, A 0, B 90, C -0, E1 0, E2 0, E3 0, E4 0} C_DIS
LIN {X 723.523, Y 0.698, Z 414, A 0, B 90, C -0, E1 0, E2 0, E3 0, E4 0} C_DIS
LIN {X 722.23, Y 2.426, Z 414, A 0, B 90, C -0, E1 0, E2 0, E3 0, E4 0} C_DIS
LIN {X 720.992, Y 4.194, Z 414, A 0, B 90, C -0, E1 0, E2 0, E3 0, E4 0} C_DIS
LIN {X 719.81, Y 6, Z 414, A 0, B 90, C -0, E1 0, E2 0, E3 0, E4 0} C_DIS
LIN {X 718.685, Y 7.842, Z 414, A 0, B 90, C -0, E1 0, E2 0, E3 0, E4 0} C_DIS
LIN {X 717.618, Y 9.719, Z 414, A 0, B 90, C -0, E1 0, E2 0, E3 0, E4 0} C_DIS
LIN {X 716.612, Y 11.628, Z 414, A 0, B 90, C -0, E1 0, E2 0, E3 0, E4 0} C_DIS
LIN {X 715.665, Y 13.568, Z 414, A 0, B 90, C -0, E1 0, E2 0, E3 0, E4 0} C_DIS
LIN {X 714.78, Y 15.536, Z 414, A 0, B 90, C -0, E1 0, E2 0, E3 0, E4 0} C_DIS
LIN {X 713.957, Y 17.532, Z 414, A 0, B 90, C -0, E1 0, E2 0, E3 0, E4 0} C_DIS
LIN {X 713.198, Y 19.552, Z 414, A 0, B 90, C -0, E1 0, E2 0, E3 0, E4 0} C_DIS
LIN {X 712.502, Y 21.595, Z 414, A 0, B 90, C -0, E1 0, E2 0, E3 0, E4 0} C_DIS
LIN {X 711.871, Y 23.659, Z 414, A 0, B 90, C -0, E1 0, E2 0, E3 0, E4 0} C_DIS
LIN {X 711.305, Y 25.742, Z 414, A 0, B 90, C -0, E1 0, E2 0, E3 0, E4 0} C_DIS
LIN {X 710.804, Y 27.841, Z 414, A 0, B 90, C -0, E1 0, E2 0, E3 0, E4 0} C_DIS
LIN {X 710.37, Y 29.956, Z 414, A 0, B 90, C -0, E1 0, E2 0, E3 0, E4 0} C_DIS
LIN {X 710.002, Y 32.082, Z 414, A 0, B 90, C -0, E1 0, E2 0, E3 0, E4 0} C_DIS
LIN {X 709.702, Y 34.22, Z 414, A 0, B 90, C -0, E1 0, E2 0, E3 0, E4 0} C_DIS
LIN {X 709.468, Y 36.366, Z 414, A 0, B 90, C -0, E1 0, E2 0, E3 0, E4 0} C_DIS
LIN {X 709.302, Y 38.518, Z 414, A 0, B 90, C -0, E1 0, E2 0, E3 0, E4 0} C_DIS
LIN {X 709.204, Y 40.674, Z 414, A 0, B 90, C -0, E1 0, E2 0, E3 0, E4 0} C_DIS
LIN {X 709.174, Y 42.832, Z 414, A 0, B 90, C -0, E1 0, E2 0, E3 0, E4 0} C_DIS
LIN {X 709.211, Y 44.99, Z 414, A 0, B 90, C -0, E1 0, E2 0, E3 0, E4 0} C_DIS
LIN {X 709.316, Y 47.146, Z 414, A 0, B 90, C -0, E1 0, E2 0, E3 0, E4 0} C_DIS
LIN {X 709.489, Y 49.297, Z 414, A 0, B 90, C -0, E1 0, E2 0, E3 0, E4 0} C_DIS
LIN {X 709.73, Y 51.442, Z 414, A 0, B 90, C -0, E1 0, E2 0, E3 0, E4 0} C_DIS
LIN {X 710.037, Y 53.578, Z 414, A 0, B 90, C -0, E1 0, E2 0, E3 0, E4 0} C_DIS
LIN {X 710.412, Y 55.704, Z 414, A 0, B 90, C -0, E1 0, E2 0, E3 0, E4 0} C_DIS
LIN {X 710.853, Y 57.817, Z 414, A 0, B 90, C -0, E1 0, E2 0, E3 0, E4 0} C_DIS
LIN {X 711.36, Y 59.915, Z 414, A 0, B 90, C -0, E1 0, E2 0, E3 0, E4 0} C_DIS
LIN {X 711.933, Y 61.996, Z 414, A 0, B 90, C -0, E1 0, E2 0, E3 0, E4 0} C_DIS
LIN {X 712.764, Y 63.456, Z 416, A 0, B 90, C -0, E1 0, E2 0, E3 0, E4 0} C_DIS
LIN {X 713.447, Y 65.491, Z 416, A 0, B 90, C -0, E1 0, E2 0, E3 0, E4 0} C_DIS
LIN {X 714.194, Y 67.503, Z 416, A 0, B 90, C -0, E1 0, E2 0, E3 0, E4 0} C_DIS
LIN {X 715.004, Y 69.492, Z 416, A 0, B 90, C -0, E1 0, E2 0, E3 0, E4 0} C_DIS
LIN {X 715.876, Y 71.453, Z 416, A 0, B 90, C -0, E1 0, E2 0, E3 0, E4 0} C_DIS
LIN {X 716.809, Y 73.387, Z 416, A 0, B 90, C -0, E1 0, E2 0, E3 0, E4 0} C_DIS
LIN {X 717.803, Y 75.29, Z 416, A 0, B 90, C -0, E1 0, E2 0, E3 0, E4 0} C_DIS
LIN {X 718.855, Y 77.161, Z 416, A 0, B 90, C -0, E1 0, E2 0, E3 0, E4 0} C_DIS
LIN {X 719.966, Y 78.998, Z 416, A 0, B 90, C -0, E1 0, E2 0, E3 0, E4 0} C_DIS
LIN {X 721.134, Y 80.799, Z 416, A 0, B 90, C -0, E1 0, E2 0, E3 0, E4 0} C_DIS
LIN {X 722.359, Y 82.563, Z 416, A 0, B 90, C -0, E1 0, E2 0, E3 0, E4 0} C_DIS
LIN {X 723.637, Y 84.287, Z 416, A 0, B 90, C -0, E1 0, E2 0, E3 0, E4 0} C_DIS
LIN {X 724.97, Y 85.97, Z 416, A 0, B 90, C -0, E1 0, E2 0, E3 0, E4 0} C_DIS
LIN {X 726.354, Y 87.611, Z 416, A 0, B 90, C -0, E1 0, E2 0, E3 0, E4 0} C_DIS
LIN {X 727.79, Y 89.207, Z 416, A 0, B 90, C -0, E1 0, E2 0, E3 0, E4 0} C_DIS
LIN {X 729.275, Y 90.758, Z 416, A 0, B 90, C -0, E1 0, E2 0, E3 0, E4 0} C_DIS
LIN {X 730.808, Y 92.261, Z 416, A 0, B 90, C -0, E1 0, E2 0, E3 0, E4 0} C_DIS
LIN {X 732.387, Y 93.715, Z 416, A 0, B 90, C -0, E1 0, E2 0, E3 0, E4 0} C_DIS
LIN {X 734.011, Y 95.119, Z 416, A 0, B 90, C -0, E1 0, E2 0, E3 0, E4 0} C_DIS
LIN {X 735.679, Y 96.471, Z 416, A 0, B 90, C -0, E1 0, E2 0, E3 0, E4 0} C_DIS
LIN {X 737.388, Y 97.77, Z 416, A 0, B 90, C -0, E1 0, E2 0, E3 0, E4 0} C_DIS
LIN {X 739.137, Y 99.014, Z 416, A 0, B 90, C -0, E1 0, E2 0, E3 0, E4 0} C_DIS
LIN {X 740.924, Y 100.204, Z 416, A 0, B 90, C -0, E1 0, E2 0, E3 0, E4 0} C_DIS
LIN {X 742.748, Y 101.336, Z 416, A 0, B 90, C -0, E1 0, E2 0, E3 0, E4 0} C_DIS
LIN {X 744.607, Y 102.411, Z 416, A 0, B 90, C -0, E1 0, E2 0, E3 0, E4 0} C_DIS
LIN {X 746.498, Y 103.426, Z 416, A 0, B 90, C -0, E1 0, E2 0, E3 0, E4 0} C_DIS
LIN {X 748.421, Y 104.382, Z 416, A 0, B 90, C -0, E1 0, E2 0, E3 0, E4 0} C_DIS
LIN {X 750.372, Y 105.277, Z 416, A 0, B 90, C -0, E1 0, E2 0, E3 0, E4 0} C_DIS
LIN {X 752.35, Y 106.11, Z 416, A 0, B 90, C -0, E1 0, E2 0, E3 0, E4 0} C_DIS
LIN {X 754.354, Y 106.881, Z 416, A 0, B 90, C -0, E1 0, E2 0, E3 0, E4 0} C_DIS
LIN {X 756.381, Y 107.588, Z 416, A 0, B 90, C -0, E1 0, E2 0, E3 0, E4 0} C_DIS
LIN {X 758.429, Y 108.231, Z 416, A 0, B 90, C -0, E1 0, E2 0, E3 0, E4 0} C_DIS
LIN {X 760.497, Y 108.81, Z 416, A 0, B 90, C -0, E1 0, E2 0, E3 0, E4 0} C_DIS
LIN {X 762.581, Y 109.323, Z 416, A 0, B 90, C -0, E1 0, E2 0, E3 0, E4 0} C_DIS
LIN {X 764.681, Y 109.771, Z 416, A 0, B 90, C -0, E1 0, E2 0, E3 0, E4 0} C_DIS
LIN {X 766.793, Y 110.153, Z 416, A 0, B 90, C -0, E1 0, E2 0, E3 0, E4 0} C_DIS
LIN {X 768.917, Y 110.468, Z 416, A 0, B 90, C -0, E1 0, E2 0, E3 0, E4 0} C_DIS
LIN {X 771.049, Y 110.716, Z 416, A 0, B 90, C -0, E1 0, E2 0, E3 0, E4 0} C_DIS
LIN {X 773.189, Y 110.897, Z 416, A 0, B 90, C -0, E1 0, E2 0, E3 0, E4 0} C_DIS
LIN {X 775.332, Y 111.01, Z 416, A 0, B 90, C -0, E1 0, E2 0, E3 0, E4 0} C_DIS
LIN {X 777.479, Y 111.057, Z 416, A 0, B 90, C -0, E1 0, E2 0, E3 0, E4 0} C_DIS
LIN {X 779.625, Y 111.036, Z 416, A 0, B 90, C -0, E1 0, E2 0, E3 0, E4 0} C_DIS
LIN {X 781.77, Y 110.947, Z 416, A 0, B 90, C -0, E1 0, E2 0, E3 0, E4 0} C_DIS
LIN {X 783.912, Y 110.791, Z 416, A 0, B 90, C -0, E1 0, E2 0, E3 0, E4 0} C_DIS
LIN {X 786.047, Y 110.568, Z 416, A 0, B 90, C -0, E1 0, E2 0, E3 0, E4 0} C_DIS
LIN {X 788.174, Y 110.278, Z 416, A 0, B 90, C -0, E1 0, E2 0, E3 0, E4 0} C_DIS
LIN {X 790.291, Y 109.922, Z 416, A 0, B 90, C -0, E1 0, E2 0, E3 0, E4 0} C_DIS
LIN {X 792.396, Y 109.499, Z 416, A 0, B 90, C -0, E1 0, E2 0, E3 0, E4 0} C_DIS
LIN {X 794.486, Y 109.01, Z 416, A 0, B 90, C -0, E1 0, E2 0, E3 0, E4 0} C_DIS
LIN {X 796.56, Y 108.455, Z 416, A 0, B 90, C -0, E1 0, E2 0, E3 0, E4 0} C_DIS
LIN {X 798.616, Y 107.836, Z 416, A 0, B 90, C -0, E1 0, E2 0, E3 0, E4 0} C_DIS
LIN {X 800.651, Y 107.153, Z 416, A 0, B 90, C -0, E1 0, E2 0, E3 0, E4 0} C_DIS
LIN {X 802.663, Y 106.406, Z 416, A 0, B 90, C -0, E1 0, E2 0, E3 0, E4 0} C_DIS
LIN {X 804.651, Y 105.596, Z 416, A 0, B 90, C -0, E1 0, E2 0, E3 0, E4 0} C_DIS
LIN {X 806.613, Y 104.724, Z 416, A 0, B 90, C -0, E1 0, E2 0, E3 0, E4 0} C_DIS
LIN {X 808.547, Y 103.791, Z 416, A 0, B 90, C -0, E1 0, E2 0, E3 0, E4 0} C_DIS
LIN {X 810.45, Y 102.797, Z 416, A 0, B 90, C -0, E1 0, E2 0, E3 0, E4 0} C_DIS
LIN {X 812.321, Y 101.745, Z 416, A 0, B 90, C -0, E1 0, E2 0, E3 0, E4 0} C_DIS
LIN {X 814.158, Y 100.634, Z 416, A 0, B 90, C -0, E1 0, E2 0, E3 0, E4 0} C_DIS
LIN {X 815.959, Y 99.466, Z 416, A 0, B 90, C -0, E1 0, E2 0, E3 0, E4 0} C_DIS
LIN {X 817.723, Y 98.241, Z 416, A 0, B 90, C -0, E1 0, E2 0, E3 0, E4 0} C_DIS
LIN {X 819.447, Y 96.963, Z 416, A 0, B 90, C -0, E1 0, E2 0, E3 0, E4 0} C_DIS
LIN {X 821.13, Y 95.63, Z 416, A 0, B 90, C -0, E1 0, E2 0, E3 0, E4 0} C_DIS
LIN {X 822.771, Y 94.246, Z 416, A 0, B 90, C -0, E1 0, E2 0, E3 0, E4 0} C_DIS
LIN {X 824.367, Y 92.81, Z 416, A 0, B 90, C -0, E1 0, E2 0, E3 0, E4 0} C_DIS
LIN {X 825.918, Y 91.325, Z 416, A 0, B 90, C -0, E1 0, E2 0, E3 0, E4 0} C_DIS
LIN {X 827.421, Y 89.792, Z 416, A 0, B 90, C -0, E1 0, E2 0, E3 0, E4 0} C_DIS
LIN {X 828.875, Y 88.213, Z 416, A 0, B 90, C -0, E1 0, E2 0, E3 0, E4 0} C_DIS
LIN {X 830.279, Y 86.589, Z 416, A 0, B 90, C -0, E1 0, E2 0, E3 0, E4 0} C_DIS
LIN {X 831.631, Y 84.921, Z 416, A 0, B 90, C -0, E1 0, E2 0, E3 0, E4 0} C_DIS
LIN {X 832.93, Y 83.212, Z 416, A 0, B 90, C -0, E1 0, E2 0, E3 0, E4 0} C_DIS
LIN {X 834.174, Y 81.463, Z 416, A 0, B 90, C -0, E1 0, E2 0, E3 0, E4 0} C_DIS
LIN {X 835.364, Y 79.675, Z 416, A 0, B 90, C -0, E1 0, E2 0, E3 0, E4 0} C_DIS
LIN {X 836.496, Y 77.852, Z 416, A 0, B 90, C -0, E1 0, E2 0, E3 0, E4 0} C_DIS
LIN {X 837.571, Y 75.993, Z 416, A 0, B 90, C -0, E1 0, E2 0, E3 0, E4 0} C_DIS
LIN {X 838.586, Y 74.102, Z 416, A 0, B 90, C -0, E1 0, E2 0, E3 0, E4 0} C_DIS
LIN {X 839.542, Y 72.179, Z 416, A 0, B 90, C -0, E1 0, E2 0, E3 0, E4 0} C_DIS
LIN {X 840.437, Y 70.228, Z 416, A 0, B 90, C -0, E1 0, E2 0, E3 0, E4 0} C_DIS
LIN {X 841.27, Y 68.25, Z 416, A 0, B 90, C -0, E1 0, E2 0, E3 0, E4 0} C_DIS
LIN {X 842.041, Y 66.246, Z 416, A 0, B 90, C -0, E1 0, E2 0, E3 0, E4 0} C_DIS
LIN {X 842.748, Y 64.219, Z 416, A 0, B 90, C -0, E1 0, E2 0, E3 0, E4 0} C_DIS
LIN {X 843.391, Y 62.171, Z 416, A 0, B 90, C -0, E1 0, E2 0, E3 0, E4 0} C_DIS
LIN {X 843.97, Y 60.103, Z 416, A 0, B 90, C -0, E1 0, E2 0, E3 0, E4 0} C_DIS
LIN {X 844.483, Y 58.019, Z 416, A 0, B 90, C -0, E1 0, E2 0, E3 0, E4 0} C_DIS
LIN {X 844.931, Y 55.919, Z 416, A 0, B 90, C -0, E1 0, E2 0, E3 0, E4 0} C_DIS
LIN {X 845.313, Y 53.807, Z 416, A 0, B 90, C -0, E1 0, E2 0, E3 0, E4 0} C_DIS
LIN {X 845.628, Y 51.683, Z 416, A 0, B 90, C -0, E1 0, E2 0, E3 0, E4 0} C_DIS
LIN {X 845.876, Y 49.551, Z 416, A 0, B 90, C -0, E1 0, E2 0, E3 0, E4 0} C_DIS
LIN {X 846.057, Y 47.411, Z 416, A 0, B 90, C -0, E1 0, E2 0, E3 0, E4 0} C_DIS
LIN {X 846.17, Y 45.268, Z 416, A 0, B 90, C -0, E1 0, E2 0, E3 0, E4 0} C_DIS
LIN {X 846.217, Y 43.121, Z 416, A 0, B 90, C -0, E1 0, E2 0, E3 0, E4 0} C_DIS
LIN {X 846.196, Y 40.975, Z 416, A 0, B 90, C -0, E1 0, E2 0, E3 0, E4 0} C_DIS
LIN {X 846.107, Y 38.83, Z 416, A 0, B 90, C -0, E1 0, E2 0, E3 0, E4 0} C_DIS
LIN {X 845.951, Y 36.688, Z 416, A 0, B 90, C -0, E1 0, E2 0, E3 0, E4 0} C_DIS
LIN {X 845.728, Y 34.553, Z 416, A 0, B 90, C -0, E1 0, E2 0, E3 0, E4 0} C_DIS
LIN {X 845.438, Y 32.426, Z 416, A 0, B 90, C -0, E1 0, E2 0, E3 0, E4 0} C_DIS
LIN {X 845.082, Y 30.309, Z 416, A 0, B 90, C -0, E1 0, E2 0, E3 0, E4 0} C_DIS
LIN {X 844.659, Y 28.204, Z 416, A 0, B 90, C -0, E1 0, E2 0, E3 0, E4 0} C_DIS
LIN {X 844.17, Y 26.114, Z 416, A 0, B 90, C -0, E1 0, E2 0, E3 0, E4 0} C_DIS
LIN {X 843.615, Y 24.04, Z 416, A 0, B 90, C -0, E1 0, E2 0, E3 0, E4 0} C_DIS
LIN {X 842.996, Y 21.984, Z 416, A 0, B 90, C -0, E1 0, E2 0, E3 0, E4 0} C_DIS
LIN {X 842.313, Y 19.949, Z 416, A 0, B 90, C -0, E1 0, E2 0, E3 0, E4 0} C_DIS
LIN {X 841.566, Y 17.937, Z 416, A 0, B 90, C -0, E1 0, E2 0, E3 0, E4 0} C_DIS
LIN {X 840.756, Y 15.948, Z 416, A 0, B 90, C -0, E1 0, E2 0, E3 0, E4 0} C_DIS
LIN {X 839.884, Y 13.987, Z 416, A 0, B 90, C -0, E1 0, E2 0, E3 0, E4 0} C_DIS
LIN {X 838.951, Y 12.053, Z 416, A 0, B 90, C -0, E1 0, E2 0, E3 0, E4 0} C_DIS
LIN {X 837.957, Y 10.15, Z 416, A 0, B 90, C -0, E1 0, E2 0, E3 0, E4 0} C_DIS
LIN {X 836.905, Y 8.279, Z 416, A 0, B 90, C -0, E1 0, E2 0, E3 0, E4 0} C_DIS
LIN {X 835.794, Y 6.442, Z 416, A 0, B 90, C -0, E1 0, E2 0, E3 0, E4 0} C_DIS
LIN {X 834.626, Y 4.641, Z 416, A 0, B 90, C -0, E1 0, E2 0, E3 0, E4 0} C_DIS
LIN {X 833.401, Y 2.877, Z 416, A 0, B 90, C -0, E1 0, E2 0, E3 0, E4 0} C_DIS
LIN {X 832.123, Y 1.153, Z 416, A 0, B 90, C -0, E1 0, E2 0, E3 0, E4 0} C_DIS
LIN {X 830.79, Y -0.53, Z 416, A 0, B 90, C -0, E1 0, E2 0, E3 0, E4 0} C_DIS
LIN {X 829.406, Y -2.171, Z 416, A 0, B 90, C -0, E1 0, E2 0, E3 0, E4 0} C_DIS
LIN {X 827.97, Y -3.767, Z 416, A 0, B 90, C -0, E1 0, E2 0, E3 0, E4 0} C_DIS
LIN {X 826.485, Y -5.318, Z 416, A 0, B 90, C -0, E1 0, E2 0, E3 0, E4 0} C_DIS
LIN {X 824.952, Y -6.821, Z 416, A 0, B 90, C -0, E1 0, E2 0, E3 0, E4 0} C_DIS
LIN {X 823.373, Y -8.275, Z 416, A 0, B 90, C -0, E1 0, E2 0, E3 0, E4 0} C_DIS
LIN {X 821.749, Y -9.679, Z 416, A 0, B 90, C -0, E1 0, E2 0, E3 0, E4 0} C_DIS
LIN {X 820.081, Y -11.031, Z 416, A 0, B 90, C -0, E1 0, E2 0, E3 0, E4 0} C_DIS
LIN {X 818.372, Y -12.33, Z 416, A 0, B 90, C -0, E1 0, E2 0, E3 0, E4 0} C_DIS
LIN {X 816.623, Y -13.574, Z 416, A 0, B 90, C -0, E1 0, E2 0, E3 0, E4 0} C_DIS
LIN {X 814.836, Y -14.764, Z 416, A 0, B 90, C -0, E1 0, E2 0, E3 0, E4 0} C_DIS
LIN {X 813.012, Y -15.896, Z 416, A 0, B 90, C -0, E1 0, E2 0, E3 0, E4 0} C_DIS
LIN {X 811.153, Y -16.971, Z 416, A 0, B 90, C -0, E1 0, E2 0, E3 0, E4 0} C_DIS
LIN {X 809.262, Y -17.986, Z 416, A 0, B 90, C -0, E1 0, E2 0, E3 0, E4 0} C_DIS
LIN {X 807.339, Y -18.942, Z 416, A 0, B 90, C -0, E1 0, E2 0, E3 0, E4 0} C_DIS
LIN {X 805.388, Y -19.837, Z 416, A 0, B 90, C -0, E1 0, E2 0, E3 0, E4 0} C_DIS
LIN {X 803.41, Y -20.67, Z 416, A 0, B 90, C -0, E1 0, E2 0, E3 0, E4 0} C_DIS
LIN {X 801.406, Y -21.441, Z 416, A 0, B 90, C -0, E1 0, E2 0, E3 0, E4 0} C_DIS
LIN {X 799.379, Y -22.148, Z 416, A 0, B 90, C -0, E1 0, E2 0, E3 0, E4 0} C_DIS
LIN {X 797.331, Y -22.791, Z 416, A 0, B 90, C -0, E1 0, E2 0, E3 0, E4 0} C_DIS
LIN {X 795.263, Y -23.37, Z 416, A 0, B 90, C -0, E1 0, E2 0, E3 0, E4 0} C_DIS
LIN {X 793.179, Y -23.883, Z 416, A 0, B 90, C -0, E1 0, E2 0, E3 0, E4 0} C_DIS
LIN {X 791.079, Y -24.331, Z 416, A 0, B 90, C -0, E1 0, E2 0, E3 0, E4 0} C_DIS
LIN {X 788.967, Y -24.713, Z 416, A 0, B 90, C -0, E1 0, E2 0, E3 0, E4 0} C_DIS
LIN {X 786.843, Y -25.028, Z 416, A 0, B 90, C -0, E1 0, E2 0, E3 0, E4 0} C_DIS
LIN {X 784.711, Y -25.276, Z 416, A 0, B 90, C -0, E1 0, E2 0, E3 0, E4 0} C_DIS
LIN {X 782.571, Y -25.457, Z 416, A 0, B 90, C -0, E1 0, E2 0, E3 0, E4 0} C_DIS
LIN {X 780.428, Y -25.57, Z 416, A 0, B 90, C -0, E1 0, E2 0, E3 0, E4 0} C_DIS
LIN {X 778.281, Y -25.617, Z 416, A 0, B 90, C -0, E1 0, E2 0, E3 0, E4 0} C_DIS
LIN {X 776.135, Y -25.596, Z 416, A 0, B 90, C -0, E1 0, E2 0, E3 0, E4 0} C_DIS
LIN {X 773.99, Y -25.507, Z 416, A 0, B 90, C -0, E1 0, E2 0, E3 0, E4 0} C_DIS
LIN {X 771.848, Y -25.351, Z 416, A 0, B 90, C -0, E1 0, E2 0, E3 0, E4 0} C_DIS
LIN {X 769.713, Y -25.128, Z 416, A 0, B 90, C -0, E1 0, E2 0, E3 0, E4 0} C_DIS
LIN {X 767.586, Y -24.838, Z 416, A 0, B 90, C -0, E1 0, E2 0, E3 0, E4 0} C_DIS
LIN {X 765.469, Y -24.482, Z 416, A 0, B 90, C -0, E1 0, E2 0, E3 0, E4 0} C_DIS
LIN {X 763.364, Y -24.059, Z 416, A 0, B 90, C -0, E1 0, E2 0, E3 0, E4 0} C_DIS
LIN {X 761.274, Y -23.57, Z 416, A 0, B 90, C -0, E1 0, E2 0, E3 0, E4 0} C_DIS
LIN {X 759.2, Y -23.015, Z 416, A 0, B 90, C -0, E1 0, E2 0, E3 0, E4 0} C_DIS
LIN {X 757.144, Y -22.396, Z 416, A 0, B 90, C -0, E1 0, E2 0, E3 0, E4 0} C_DIS
LIN {X 755.109, Y -21.713, Z 416, A 0, B 90, C -0, E1 0, E2 0, E3 0, E4 0} C_DIS
LIN {X 753.097, Y -20.966, Z 416, A 0, B 90, C -0, E1 0, E2 0, E3 0, E4 0} C_DIS
LIN {X 751.109, Y -20.156, Z 416, A 0, B 90, C -0, E1 0, E2 0, E3 0, E4 0} C_DIS
LIN {X 749.147, Y -19.284, Z 416, A 0, B 90, C -0, E1 0, E2 0, E3 0, E4 0} C_DIS
LIN {X 747.213, Y -18.351, Z 416, A 0, B 90, C -0, E1 0, E2 0, E3 0, E4 0} C_DIS
LIN {X 745.31, Y -17.357, Z 416, A 0, B 90, C -0, E1 0, E2 0, E3 0, E4 0} C_DIS
LIN {X 743.439, Y -16.305, Z 416, A 0, B 90, C -0, E1 0, E2 0, E3 0, E4 0} C_DIS
LIN {X 741.602, Y -15.194, Z 416, A 0, B 90, C -0, E1 0, E2 0, E3 0, E4 0} C_DIS
LIN {X 739.801, Y -14.026, Z 416, A 0, B 90, C -0, E1 0, E2 0, E3 0, E4 0} C_DIS
LIN {X 738.037, Y -12.801, Z 416, A 0, B 90, C -0, E1 0, E2 0, E3 0, E4 0} C_DIS
LIN {X 736.313, Y -11.523, Z 416, A 0, B 90, C -0, E1 0, E2 0, E3 0, E4 0} C_DIS
LIN {X 734.63, Y -10.19, Z 416, A 0, B 90, C -0, E1 0, E2 0, E3 0, E4 0} C_DIS
LIN {X 732.989, Y -8.806, Z 416, A 0, B 90, C -0, E1 0, E2 0, E3 0, E4 0} C_DIS
LIN {X 731.393, Y -7.37, Z 416, A 0, B 90, C -0, E1 0, E2 0, E3 0, E4 0} C_DIS
LIN {X 729.842, Y -5.885, Z 416, A 0, B 90, C -0, E1 0, E2 0, E3 0, E4 0} C_DIS
LIN {X 728.339, Y -4.352, Z 416, A 0, B 90, C -0, E1 0, E2 0, E3 0, E4 0} C_DIS
LIN {X 726.885, Y -2.773, Z 416, A 0, B 90, C -0, E1 0, E2 0, E3 0, E4 0} C_DIS
LIN {X 725.481, Y -1.149, Z 416, A 0, B 90, C -0, E1 0, E2 0, E3 0, E4 0} C_DIS
LIN {X 724.129, Y 0.519, Z 416, A 0, B 90, C -0, E1 0, E2 0, E3 0, E4 0} C_DIS
LIN {X 722.83, Y 2.228, Z 416, A 0, B 90, C -0, E1 0, E2 0, E3 0, E4 0} C_DIS
LIN {X 721.586, Y 3.977, Z 416, A 0, B 90, C -0, E1 0, E2 0, E3 0, E4 0} C_DIS
LIN {X 720.396, Y 5.765, Z 416, A 0, B 90, C -0, E1 0, E2 0, E3 0, E4 0} C_DIS
LIN {X 719.264, Y 7.588, Z 416, A 0, B 90, C -0, E1 0, E2 0, E3 0, E4 0} C_DIS
LIN {X 718.189, Y 9.447, Z 416, A 0, B 90, C -0, E1 0, E2 0, E3 0, E4 0} C_DIS
LIN {X 717.174, Y 11.338, Z 416, A 0, B 90, C -0, E1 0, E2 0, E3 0, E4 0} C_DIS
LIN {X 716.218, Y 13.261, Z 416, A 0, B 90, C -0, E1 0, E2 0, E3 0, E4 0} C_DIS
LIN {X 715.323, Y 15.212, Z 416, A 0, B 90, C -0, E1 0, E2 0, E3 0, E4 0} C_DIS
LIN {X 714.49, Y 17.19, Z 416, A 0, B 90, C -0, E1 0, E2 0, E3 0, E4 0} C_DIS
LIN {X 713.719, Y 19.194, Z 416, A 0, B 90, C -0, E1 0, E2 0, E3 0, E4 0} C_DIS
LIN {X 713.012, Y 21.221, Z 416, A 0, B 90, C -0, E1 0, E2 0, E3 0, E4 0} C_DIS
LIN {X 712.369, Y 23.269, Z 416, A 0, B 90, C -0, E1 0, E2 0, E3 0, E4 0} C_DIS
LIN {X 711.79, Y 25.337, Z 416, A 0, B 90, C -0, E1 0, E2 0, E3 0, E4 0} C_DIS
LIN {X 711.277, Y 27.421, Z 416, A 0, B 90, C -0, E1 0, E2 0, E3 0, E4 0} C_DIS
LIN {X 710.829, Y 29.521, Z 416, A 0, B 90, C -0, E1 0, E2 0, E3 0, E4 0} C_DIS
LIN {X 710.447, Y 31.633, Z 416, A 0, B 90, C -0, E1 0, E2 0, E3 0, E4 0} C_DIS
LIN {X 710.132, Y 33.757, Z 416, A 0, B 90, C -0, E1 0, E2 0, E3 0, E4 0} C_DIS
LIN {X 709.884, Y 35.889, Z 416, A 0, B 90, C -0, E1 0, E2 0, E3 0, E4 0} C_DIS
LIN {X 709.703, Y 38.029, Z 416, A 0, B 90, C -0, E1 0, E2 0, E3 0, E4 0} C_DIS
LIN {X 709.59, Y 40.172, Z 416, A 0, B 90, C -0, E1 0, E2 0, E3 0, E4 0} C_DIS
LIN {X 709.543, Y 42.319, Z 416, A 0, B 90, C -0, E1 0, E2 0, E3 0, E4 0} C_DIS
